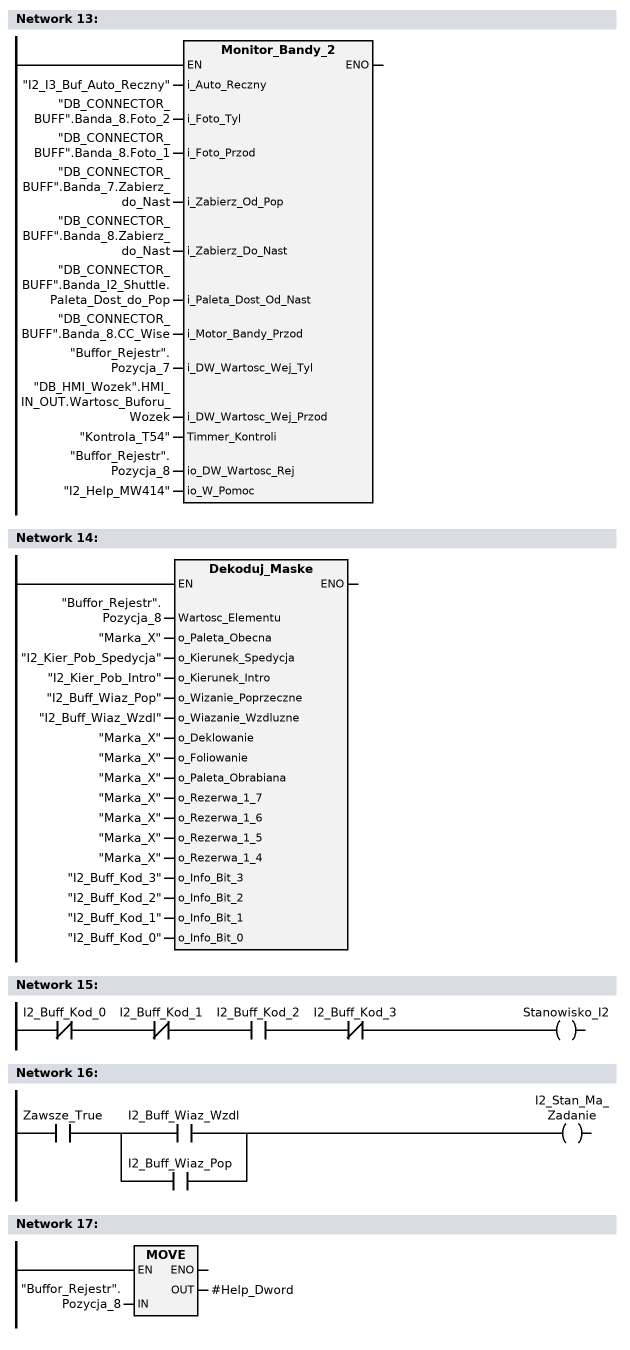
[picture p225: Stan_Intro_Pob_I2 networks 13-17]
NETWORK
TITLE =
//Monitoring band 8
//
      CALL  "Monitor_Bandy_2" (
           i_Auto_Reczny            := "I2_I3_Buf_Auto_Reczny",
           i_Foto_Tyl               := "DB_CONNECTOR_BUFF".Banda_8.Foto_2,
           i_Foto_Przod             := "DB_CONNECTOR_BUFF".Banda_8.Foto_1,
           i_Zabierz_Od_Pop         := "DB_CONNECTOR_BUFF".Banda_7.Zabierz_do_Nast,
           i_Zabierz_Do_Nast        := "DB_CONNECTOR_BUFF".Banda_8.Zabierz_do_Nast,
           i_Paleta_Dost_Od_Nast    := "DB_CONNECTOR_BUFF".Banda_I2_Shuttle.Paleta_Dost_do_Pop,
           i_Motor_Bandy_Przod      := "DB_CONNECTOR_BUFF".Banda_8.CC_Wise,
           i_DW_Wartosc_Wej_Tyl     := "Buffor_Rejestr".Pozycja_7,
           i_DW_Wartosc_Wej_Przod   := "DB_HMI_Wozek".HMI_IN_OUT.Wartosc_Buforu_Wozek,
           Timmer_Kontroli          := "Kontrola_T54",
           io_DW_Wartosc_Rej        := "Buffor_Rejestr".Pozycja_8,
           io_W_Pomoc               := "I2_Help_MW414");
NETWORK
TITLE =
//Dekouj maske
//Potrzebne do okreslenia kierunku kursu
      CALL  "Dekoduj_Maske" (
           Wartosc_Elementu         := "Buffor_Rejestr".Pozycja_8,
           o_Paleta_Obecna          := "Marka_X",
           o_Kierunek_Spedycja      := "I2_Kier_Pob_Spedycja",
           o_Kierunek_Intro         := "I2_Kier_Pob_Intro",
           o_Wizanie_Poprzeczne     := "I2_Buff_Wiaz_Pop",
           o_Wiazanie_Wzdluzne      := "I2_Buff_Wiaz_Wzdl",
           o_Deklowanie             := "Marka_X",
           o_Foliowanie             := "Marka_X",
           o_Paleta_Obrabiana       := "Marka_X",
           o_Rezerwa_1_7            := "Marka_X",
           o_Rezerwa_1_6            := "Marka_X",
           o_Rezerwa_1_5            := "Marka_X",
           o_Rezerwa_1_4            := "Marka_X",
           o_Info_Bit_3             := "I2_Buff_Kod_3",
           o_Info_Bit_2             := "I2_Buff_Kod_2",
           o_Info_Bit_1             := "I2_Buff_Kod_1",
           o_Info_Bit_0             := "I2_Buff_Kod_0");
NETWORK
TITLE =
//Stanowisko intro kod 
      AN    "I2_Buff_Kod_0";
      AN    "I2_Buff_Kod_1";
      A     "I2_Buff_Kod_2";
      AN    "I2_Buff_Kod_3";
      =     "Stanowisko_I2";
NETWORK
TITLE =
//Stanowisko intro ma jakies zadanie
      A     "Zawsze_True";
      A(;
      O     "I2_Buff_Wiaz_Wzdl";
      O     "I2_Buff_Wiaz_Pop";
      );
      =     "I2_Stan_Ma_Zadanie";
NETWORK
TITLE =
      L     "Buffor_Rejestr".Pozycja_8;
      T     #Help_Dword;
      NOP   0;
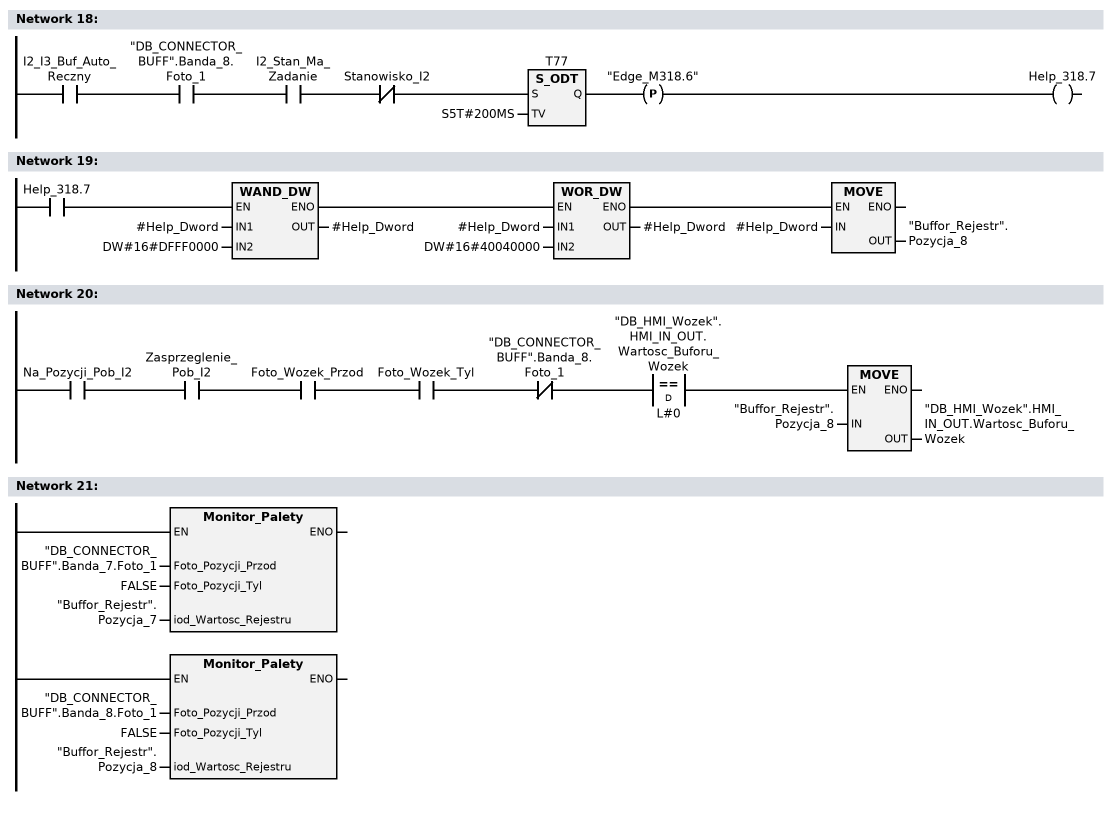
NETWORK
TITLE =
//Przepisanie wartosci nowej wartosci kodu jesli jest zadanie a paleta nie znana
//Domyslnie wysylana jest na Gender
      A(;
      A     "I2_I3_Buf_Auto_Reczny";
      A     "DB_CONNECTOR_BUFF".Banda_8.Foto_1;
      A     "I2_Stan_Ma_Zadanie";
      AN    "Stanowisko_I2";
      L     S5T#200MS;
      SD    "T77";
      NOP   0;
      NOP   0;
      NOP   0;
      A     "T77";
      );
      FP    "Edge_M318.6";
      =     "Help_318.7";
NETWORK
TITLE =
//Przypisanie nowej wartosci do palety
      A(;
      A(;
      A     "Help_318.7";
      JNB   _003;
      L     #Help_Dword;
      L     DW#16#DFFF0000;
      AD;
      T     #Help_Dword;
      SET;
      SAVE;
      CLR;
_003: A     BR;
      );
      JNB   _004;
      L     #Help_Dword;
      L     DW#16#40040000;
      OD;
      T     #Help_Dword;
      SET;
      SAVE;
      CLR;
_004: A     BR;
      );
      JNB   _005;
      L     #Help_Dword;
      T     "Buffor_Rejestr".Pozycja_8;
_005: NOP   0;
NETWORK
TITLE =
//db128.db208 -wartosc rejestru na wozka
      A     "Na_Pozycji_Pob_I2";
      A     "Zasprzeglenie_Pob_I2";
      A     "Foto_Wozek_Przod";
      A     "Foto_Wozek_Tyl";
      AN    "DB_CONNECTOR_BUFF".Banda_8.Foto_1;
      A(;
      L     "DB_HMI_Wozek".HMI_IN_OUT.Wartosc_Buforu_Wozek;
      L     L#0;
      ==D;
      );
      JNB   _006;
      L     "Buffor_Rejestr".Pozycja_8;
      T     "DB_HMI_Wozek".HMI_IN_OUT.Wartosc_Buforu_Wozek;
_006: NOP   0;
NETWORK
TITLE =
//Monitor palet
      CALL  "Monitor_Palety" (
           Foto_Pozycji_Przod       := "DB_CONNECTOR_BUFF".Banda_7.Foto_1,
           Foto_Pozycji_Tyl         := FALSE,
           iod_Wartosc_Rejestru     := "Buffor_Rejestr".Pozycja_7);
      CALL  "Monitor_Palety" (
           Foto_Pozycji_Przod       := "DB_CONNECTOR_BUFF".Banda_8.Foto_1,
           Foto_Pozycji_Tyl         := FALSE,
           iod_Wartosc_Rejestru     := "Buffor_Rejestr".Pozycja_8);
END_FUNCTION_BLOCK

FUNCTION_BLOCK "Stan_Intro_Pob_I3"	// FB 9
//Stanowisko intro Pobieranie
//Linia zlozona z 5 band odbierajacych
//
//
//B7 B8 BW
//===>
//
//2 Bandy kierunek zgodny
VERSION : 0.1
VAR
  Banda_17 : FB 33;
  Banda_18 : FB 33;
END_VAR
VAR_TEMP
  Help_Bit_1 : BOOL ;
  Help_Reczny : BOOL ;
  Help_int : INT ;
  Help_Dword : DWORD ;
  Help_INT_1 : DINT ;
END_VAR
BEGIN
NETWORK
TITLE =
//Ten Network celowo jest wolny
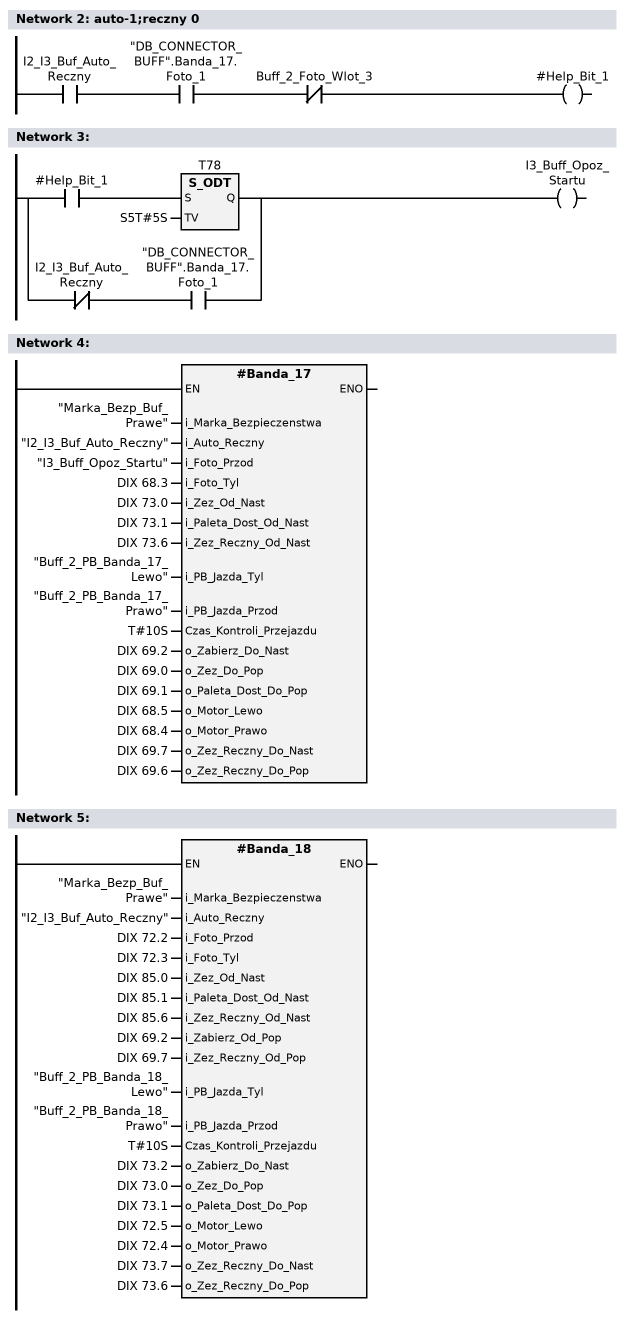
NETWORK
TITLE = auto-1;reczny 0
      A     "I2_I3_Buf_Auto_Reczny";
      A     "DB_CONNECTOR_BUFF".Banda_17.Foto_1;
      AN    "Buff_2_Foto_Wlot_3";
      =     #Help_Bit_1;
NETWORK
TITLE =
//Opoznienie startu po polozeniu palety
//
      O(;
      A     #Help_Bit_1;
      L     S5T#5S;
      SD    "T78";
      NOP   0;
      NOP   0;
      NOP   0;
      A     "T78";
      );
      O;
      AN    "I2_I3_Buf_Auto_Reczny";
      A     "DB_CONNECTOR_BUFF".Banda_17.Foto_1;
      =     "I3_Buff_Opoz_Startu";
NETWORK
TITLE =
//Banda 7
      CALL  #Banda_17 (
           i_Marka_Bezpieczenstwa   := "Marka_Bezp_Buf_Prawe",
           i_Auto_Reczny            := "I2_I3_Buf_Auto_Reczny",
           i_Foto_Przod             := "I3_Buff_Opoz_Startu",
           i_Foto_Tyl               := DIX 68.3,
           i_Zez_Od_Nast            := DIX 73.0,
           i_Paleta_Dost_Od_Nast    := DIX 73.1,
           i_Zez_Reczny_Od_Nast     := DIX 73.6,
           i_PB_Jazda_Tyl           := "Buff_2_PB_Banda_17_Lewo",
           i_PB_Jazda_Przod         := "Buff_2_PB_Banda_17_Prawo",
           Czas_Kontroli_Przejazdu  := T#10S,
           o_Zabierz_Do_Nast        := DIX 69.2,
           o_Zez_Do_Pop             := DIX 69.0,
           o_Paleta_Dost_Do_Pop     := DIX 69.1,
           o_Motor_Lewo             := DIX 68.5,
           o_Motor_Prawo            := DIX 68.4,
           o_Zez_Reczny_Do_Nast     := DIX 69.7,
           o_Zez_Reczny_Do_Pop      := DIX 69.6);
NETWORK
TITLE =
//Banda 8
      CALL  #Banda_18 (
           i_Marka_Bezpieczenstwa   := "Marka_Bezp_Buf_Prawe",
           i_Auto_Reczny            := "I2_I3_Buf_Auto_Reczny",
           i_Foto_Przod             := DIX 72.2,
           i_Foto_Tyl               := DIX 72.3,
           i_Zez_Od_Nast            := DIX 85.0,
           i_Paleta_Dost_Od_Nast    := DIX 85.1,
           i_Zez_Reczny_Od_Nast     := DIX 85.6,
           i_Zabierz_Od_Pop         := DIX 69.2,
           i_Zez_Reczny_Od_Pop      := DIX 69.7,
           i_PB_Jazda_Tyl           := "Buff_2_PB_Banda_18_Lewo",
           i_PB_Jazda_Przod         := "Buff_2_PB_Banda_18_Prawo",
           Czas_Kontroli_Przejazdu  := T#10S,
           o_Zabierz_Do_Nast        := DIX 73.2,
           o_Zez_Do_Pop             := DIX 73.0,
           o_Paleta_Dost_Do_Pop     := DIX 73.1,
           o_Motor_Lewo             := DIX 72.5,
           o_Motor_Prawo            := DIX 72.4,
           o_Zez_Reczny_Do_Nast     := DIX 73.7,
           o_Zez_Reczny_Do_Pop      := DIX 73.6);
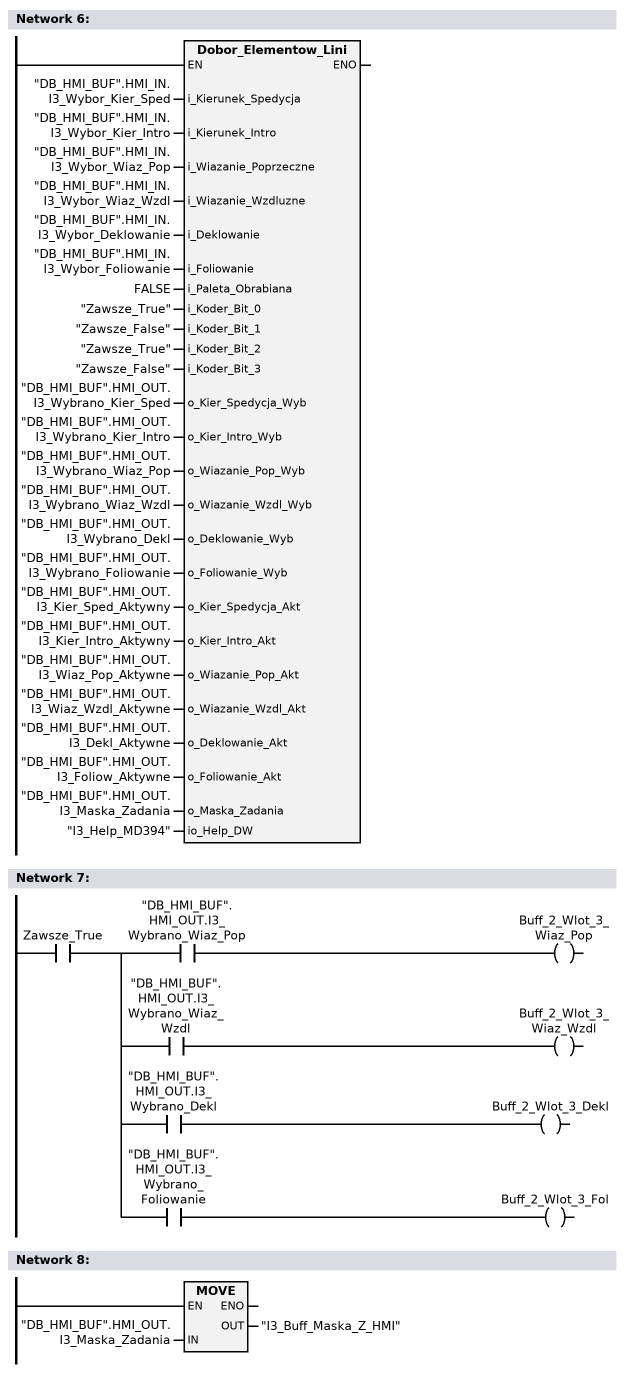
NETWORK
TITLE =
//Wybor Elementow na lini koder nr 5
      CALL  "Dobor_Elementow_Lini" (
           i_Kierunek_Spedycja      := "DB_HMI_BUF".HMI_IN.I3_Wybor_Kier_Sped,
           i_Kierunek_Intro         := "DB_HMI_BUF".HMI_IN.I3_Wybor_Kier_Intro,
           i_Wiazanie_Poprzeczne    := "DB_HMI_BUF".HMI_IN.I3_Wybor_Wiaz_Pop,
           i_Wiazanie_Wzdluzne      := "DB_HMI_BUF".HMI_IN.I3_Wybor_Wiaz_Wzdl,
           i_Deklowanie             := "DB_HMI_BUF".HMI_IN.I3_Wybor_Deklowanie,
           i_Foliowanie             := "DB_HMI_BUF".HMI_IN.I3_Wybor_Foliowanie,
           i_Paleta_Obrabiana       := FALSE,
           i_Koder_Bit_0            := "Zawsze_True",
           i_Koder_Bit_1            := "Zawsze_False",
           i_Koder_Bit_2            := "Zawsze_True",
           i_Koder_Bit_3            := "Zawsze_False",
           o_Kier_Spedycja_Wyb      := "DB_HMI_BUF".HMI_OUT.I3_Wybrano_Kier_Sped,
           o_Kier_Intro_Wyb         := "DB_HMI_BUF".HMI_OUT.I3_Wybrano_Kier_Intro,
           o_Wiazanie_Pop_Wyb       := "DB_HMI_BUF".HMI_OUT.I3_Wybrano_Wiaz_Pop,
           o_Wiazanie_Wzdl_Wyb      := "DB_HMI_BUF".HMI_OUT.I3_Wybrano_Wiaz_Wzdl,
           o_Deklowanie_Wyb         := "DB_HMI_BUF".HMI_OUT.I3_Wybrano_Dekl,
           o_Foliowanie_Wyb         := "DB_HMI_BUF".HMI_OUT.I3_Wybrano_Foliowanie,
           o_Kier_Spedycja_Akt      := "DB_HMI_BUF".HMI_OUT.I3_Kier_Sped_Aktywny,
           o_Kier_Intro_Akt         := "DB_HMI_BUF".HMI_OUT.I3_Kier_Intro_Aktywny,
           o_Wiazanie_Pop_Akt       := "DB_HMI_BUF".HMI_OUT.I3_Wiaz_Pop_Aktywne,
           o_Wiazanie_Wzdl_Akt      := "DB_HMI_BUF".HMI_OUT.I3_Wiaz_Wzdl_Aktywne,
           o_Deklowanie_Akt         := "DB_HMI_BUF".HMI_OUT.I3_Dekl_Aktywne,
           o_Foliowanie_Akt         := "DB_HMI_BUF".HMI_OUT.I3_Foliow_Aktywne,
           o_Maska_Zadania          := "DB_HMI_BUF".HMI_OUT.I3_Maska_Zadania,
           io_Help_DW               := "I3_Help_MD394");
NETWORK
TITLE =
//Wyswietlenie lampek zadania lini
      A     "Zawsze_True";
      =     L 12.0;
      A     L 12.0;
      A     "DB_HMI_BUF".HMI_OUT.I3_Wybrano_Wiaz_Pop;
      =     "Buff_2_Wlot_3_Wiaz_Pop";
      A     L 12.0;
      A     "DB_HMI_BUF".HMI_OUT.I3_Wybrano_Wiaz_Wzdl;
      =     "Buff_2_Wlot_3_Wiaz_Wzdl";
      A     L 12.0;
      A     "DB_HMI_BUF".HMI_OUT.I3_Wybrano_Dekl;
      =     "Buff_2_Wlot_3_Dekl";
      A     L 12.0;
      A     "DB_HMI_BUF".HMI_OUT.I3_Wybrano_Foliowanie;
      =     "Buff_2_Wlot_3_Fol";
NETWORK
TITLE =
//Przypisanie maski zadania do bandy wejsciowej
      L     "DB_HMI_BUF".HMI_OUT.I3_Maska_Zadania;
      T     "I3_Buff_Maska_Z_HMI";
      NOP   0;
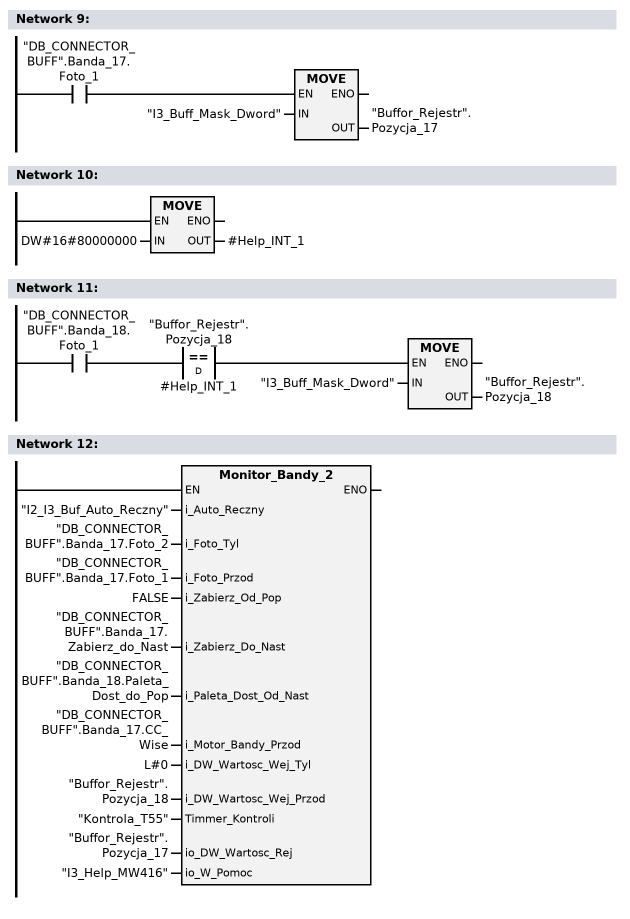
NETWORK
TITLE =
//Zbudowanie z maski podwojnego slowa
      A     "DB_CONNECTOR_BUFF".Banda_17.Foto_1;
      JNB   _001;
      L     "I3_Buff_Mask_Dword";
      T     "Buffor_Rejestr".Pozycja_17;
_001: NOP   0;
NETWORK
TITLE =
      L     DW#16#80000000;
      T     #Help_INT_1;
      NOP   0;
NETWORK
TITLE =
//sprawdzenie dla fotokomorki bandy 8
      A     "DB_CONNECTOR_BUFF".Banda_18.Foto_1;
      A(;
      L     "Buffor_Rejestr".Pozycja_18;
      L     #Help_INT_1;
      ==D;
      );
      JNB   _002;
      L     "I3_Buff_Mask_Dword";
      T     "Buffor_Rejestr".Pozycja_18;
_002: NOP   0;
NETWORK
TITLE =
//Monitoring band 7
      CALL  "Monitor_Bandy_2" (
           i_Auto_Reczny            := "I2_I3_Buf_Auto_Reczny",
           i_Foto_Tyl               := "DB_CONNECTOR_BUFF".Banda_17.Foto_2,
           i_Foto_Przod             := "DB_CONNECTOR_BUFF".Banda_17.Foto_1,
           i_Zabierz_Od_Pop         := FALSE,
           i_Zabierz_Do_Nast        := "DB_CONNECTOR_BUFF".Banda_17.Zabierz_do_Nast,
           i_Paleta_Dost_Od_Nast    := "DB_CONNECTOR_BUFF".Banda_18.Paleta_Dost_do_Pop,
           i_Motor_Bandy_Przod      := "DB_CONNECTOR_BUFF".Banda_17.CC_Wise,
           i_DW_Wartosc_Wej_Tyl     := L#0,
           i_DW_Wartosc_Wej_Przod   := "Buffor_Rejestr".Pozycja_18,
           Timmer_Kontroli          := "Kontrola_T55",
           io_DW_Wartosc_Rej        := "Buffor_Rejestr".Pozycja_17,
           io_W_Pomoc               := "I3_Help_MW416");
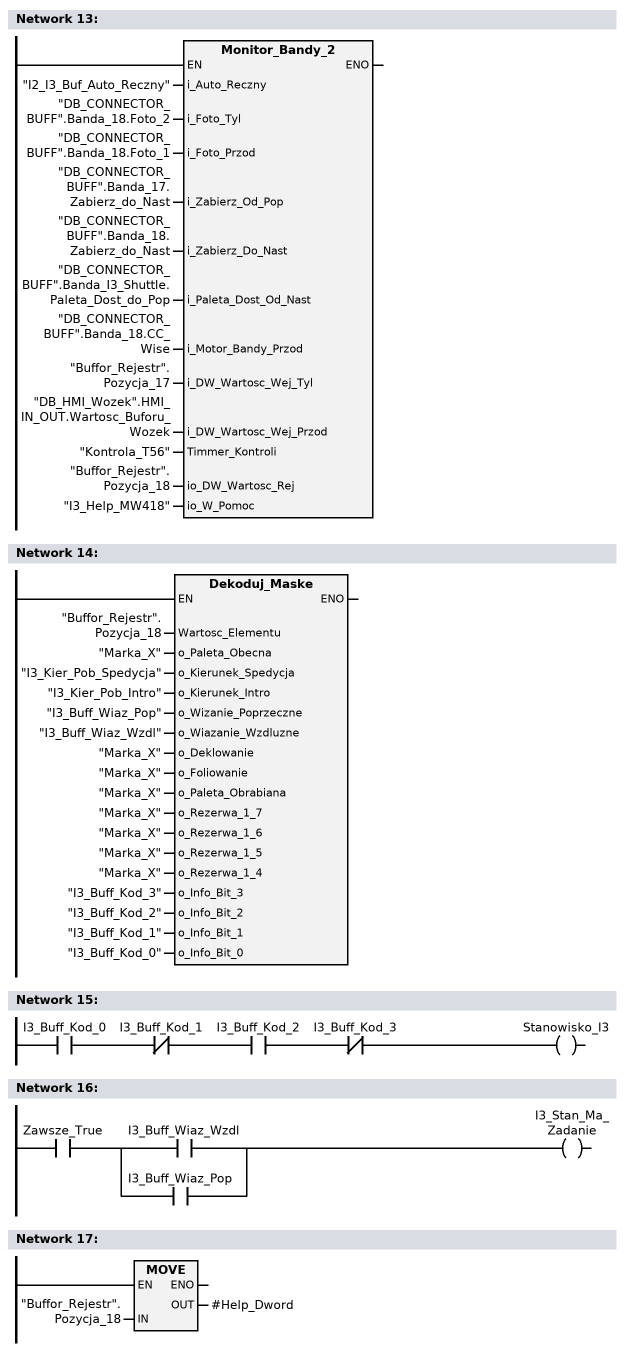
NETWORK
TITLE =
//Monitoring band 8
//
      CALL  "Monitor_Bandy_2" (
           i_Auto_Reczny            := "I2_I3_Buf_Auto_Reczny",
           i_Foto_Tyl               := "DB_CONNECTOR_BUFF".Banda_18.Foto_2,
           i_Foto_Przod             := "DB_CONNECTOR_BUFF".Banda_18.Foto_1,
           i_Zabierz_Od_Pop         := "DB_CONNECTOR_BUFF".Banda_17.Zabierz_do_Nast,
           i_Zabierz_Do_Nast        := "DB_CONNECTOR_BUFF".Banda_18.Zabierz_do_Nast,
           i_Paleta_Dost_Od_Nast    := "DB_CONNECTOR_BUFF".Banda_I3_Shuttle.Paleta_Dost_do_Pop,
           i_Motor_Bandy_Przod      := "DB_CONNECTOR_BUFF".Banda_18.CC_Wise,
           i_DW_Wartosc_Wej_Tyl     := "Buffor_Rejestr".Pozycja_17,
           i_DW_Wartosc_Wej_Przod   := "DB_HMI_Wozek".HMI_IN_OUT.Wartosc_Buforu_Wozek,
           Timmer_Kontroli          := "Kontrola_T56",
           io_DW_Wartosc_Rej        := "Buffor_Rejestr".Pozycja_18,
           io_W_Pomoc               := "I3_Help_MW418");
NETWORK
TITLE =
//Dekouj maske
//Potrzebne do okreslenia kierunku kursu
      CALL  "Dekoduj_Maske" (
           Wartosc_Elementu         := "Buffor_Rejestr".Pozycja_18,
           o_Paleta_Obecna          := "Marka_X",
           o_Kierunek_Spedycja      := "I3_Kier_Pob_Spedycja",
           o_Kierunek_Intro         := "I3_Kier_Pob_Intro",
           o_Wizanie_Poprzeczne     := "I3_Buff_Wiaz_Pop",
           o_Wiazanie_Wzdluzne      := "I3_Buff_Wiaz_Wzdl",
           o_Deklowanie             := "Marka_X",
           o_Foliowanie             := "Marka_X",
           o_Paleta_Obrabiana       := "Marka_X",
           o_Rezerwa_1_7            := "Marka_X",
           o_Rezerwa_1_6            := "Marka_X",
           o_Rezerwa_1_5            := "Marka_X",
           o_Rezerwa_1_4            := "Marka_X",
           o_Info_Bit_3             := "I3_Buff_Kod_3",
           o_Info_Bit_2             := "I3_Buff_Kod_2",
           o_Info_Bit_1             := "I3_Buff_Kod_1",
           o_Info_Bit_0             := "I3_Buff_Kod_0");
NETWORK
TITLE =
//Stanowisko intro kod 
      A     "I3_Buff_Kod_0";
      AN    "I3_Buff_Kod_1";
      A     "I3_Buff_Kod_2";
      AN    "I3_Buff_Kod_3";
      =     "Stanowisko_I3";
NETWORK
TITLE =
//Stanowisko intro ma jakies zadanie
      A     "Zawsze_True";
      A(;
      O     "I3_Buff_Wiaz_Wzdl";
      O     "I3_Buff_Wiaz_Pop";
      );
      =     "I3_Stan_Ma_Zadanie";
NETWORK
TITLE =
      L     "Buffor_Rejestr".Pozycja_18;
      T     #Help_Dword;
      NOP   0;
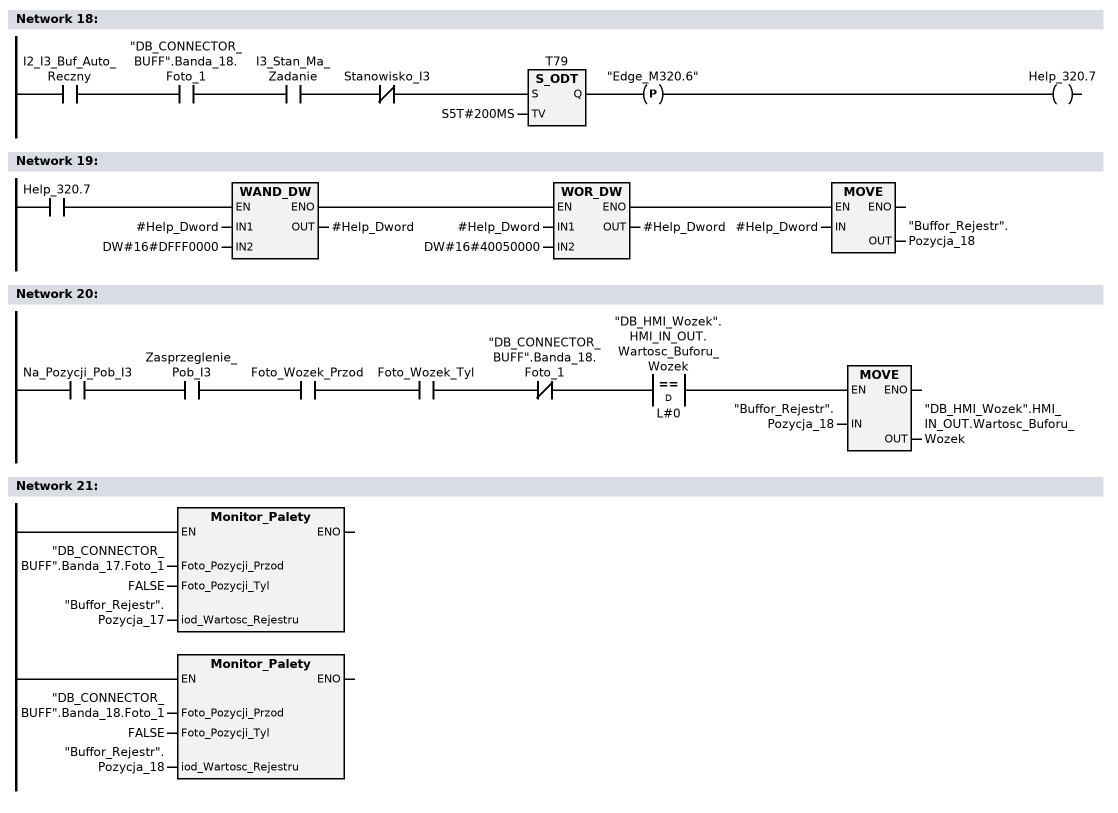
NETWORK
TITLE =
//Przepisanie wartosci nowej wartosci kodu jesli jest zadanie a paleta nie znana
//Domyslnie wysylana jest na Gender
      A(;
      A     "I2_I3_Buf_Auto_Reczny";
      A     "DB_CONNECTOR_BUFF".Banda_18.Foto_1;
      A     "I3_Stan_Ma_Zadanie";
      AN    "Stanowisko_I3";
      L     S5T#200MS;
      SD    "T79";
      NOP   0;
      NOP   0;
      NOP   0;
      A     "T79";
      );
      FP    "Edge_M320.6";
      =     "Help_320.7";
NETWORK
TITLE =
//Przypisanie nowej wartosci do palety
      A(;
      A(;
      A     "Help_320.7";
      JNB   _003;
      L     #Help_Dword;
      L     DW#16#DFFF0000;
      AD;
      T     #Help_Dword;
      SET;
      SAVE;
      CLR;
_003: A     BR;
      );
      JNB   _004;
      L     #Help_Dword;
      L     DW#16#40050000;
      OD;
      T     #Help_Dword;
      SET;
      SAVE;
      CLR;
_004: A     BR;
      );
      JNB   _005;
      L     #Help_Dword;
      T     "Buffor_Rejestr".Pozycja_18;
_005: NOP   0;
NETWORK
TITLE =
//db128.db208 -wartosc rejestru na wozka
      A     "Na_Pozycji_Pob_I3";
      A     "Zasprzeglenie_Pob_I3";
      A     "Foto_Wozek_Przod";
      A     "Foto_Wozek_Tyl";
      AN    "DB_CONNECTOR_BUFF".Banda_18.Foto_1;
      A(;
      L     "DB_HMI_Wozek".HMI_IN_OUT.Wartosc_Buforu_Wozek;
      L     L#0;
      ==D;
      );
      JNB   _006;
      L     "Buffor_Rejestr".Pozycja_18;
      T     "DB_HMI_Wozek".HMI_IN_OUT.Wartosc_Buforu_Wozek;
_006: NOP   0;
NETWORK
TITLE =
//Monitor palet
      CALL  "Monitor_Palety" (
           Foto_Pozycji_Przod       := "DB_CONNECTOR_BUFF".Banda_17.Foto_1,
           Foto_Pozycji_Tyl         := FALSE,
           iod_Wartosc_Rejestru     := "Buffor_Rejestr".Pozycja_17);
      CALL  "Monitor_Palety" (
           Foto_Pozycji_Przod       := "DB_CONNECTOR_BUFF".Banda_18.Foto_1,
           Foto_Pozycji_Tyl         := FALSE,
           iod_Wartosc_Rejestru     := "Buffor_Rejestr".Pozycja_18);
END_FUNCTION_BLOCK

FUNCTION_BLOCK "FB_Uzbrajanie"	// FB 10
//Funkcja odpowiada za sterowanie uzbrajaniem palety.
//Gdy jest stan wysoki na wejsciu uzbrajanie palety to aktywne jest przycisk 
//PB_uzbrajanie (Pojedyncze klikniecie). Aby zakonczyc uzbrajanie nalezy wcisnac 
//przycisk dwukrotnie w krotkim czasie.
VERSION : 0.1
VAR_INPUT
  i_Tryb_Uzbrajania : BOOL ;
  i_Zezw_Na_Uzb : BOOL ;	//Zezwolenie na uzbrajanie
  i_PB_Uzbrajanie : BOOL ;	//Przycisk grzybkowy uzbrajania
  i_PB_Wybor_O_Lewo : BOOL ;	//Wybor obrot w lewa strone
  i_PB_Wybor_O_Prawo : BOOL ;	//Wybor obrot w prawa strone
  i_Pedal_Zal : BOOL ;	//Wlaczenie pedala
  t_Czas_Kontrolny : TIME ;
  t_Czas_Konca : TIME ;
END_VAR
VAR_OUTPUT
  o_Oczekiwanie_Aktywne : BOOL ;
  o_Lampka_Uzb_Lewo : BOOL ;
  o_Lampka_Uzb_Prawo : BOOL ;
  o_Sygnal_Startu_Uzbr : BOOL ;	//Sygnal krotki startu uzbrajania
  o_Sygnal_Kon_Uzbr : BOOL ;	//Sygnal konca uzbrajania
  o_Pedal_Lewo : BOOL ;
  o_Pedal_Prawo : BOOL ;
END_VAR
VAR_IN_OUT
  io_Uzbrajanie_W_Trakcie : BOOL ;
END_VAR
VAR
  Czas_Kontrolny : SFB 4;	//Czas kontrolny przycisku
  Czas_Konca : SFB 4;
  Edge_1 : BOOL ;
  Edge_2 : BOOL ;
  Edge_3 : BOOL ;
  Help_Timer : BOOL ;
  H_Uzbrajanie_W_Trakcie : BOOL ;
  H_Lewo_Prawo : BOOL ;	//0-Lewo;1-Prawo
END_VAR
VAR_TEMP
  Temp_Bit_1 : BOOL ;
  Temp_Bit_2 : BOOL ;
END_VAR
BEGIN
NETWORK
TITLE =
//Ten Network celowo jest wolny
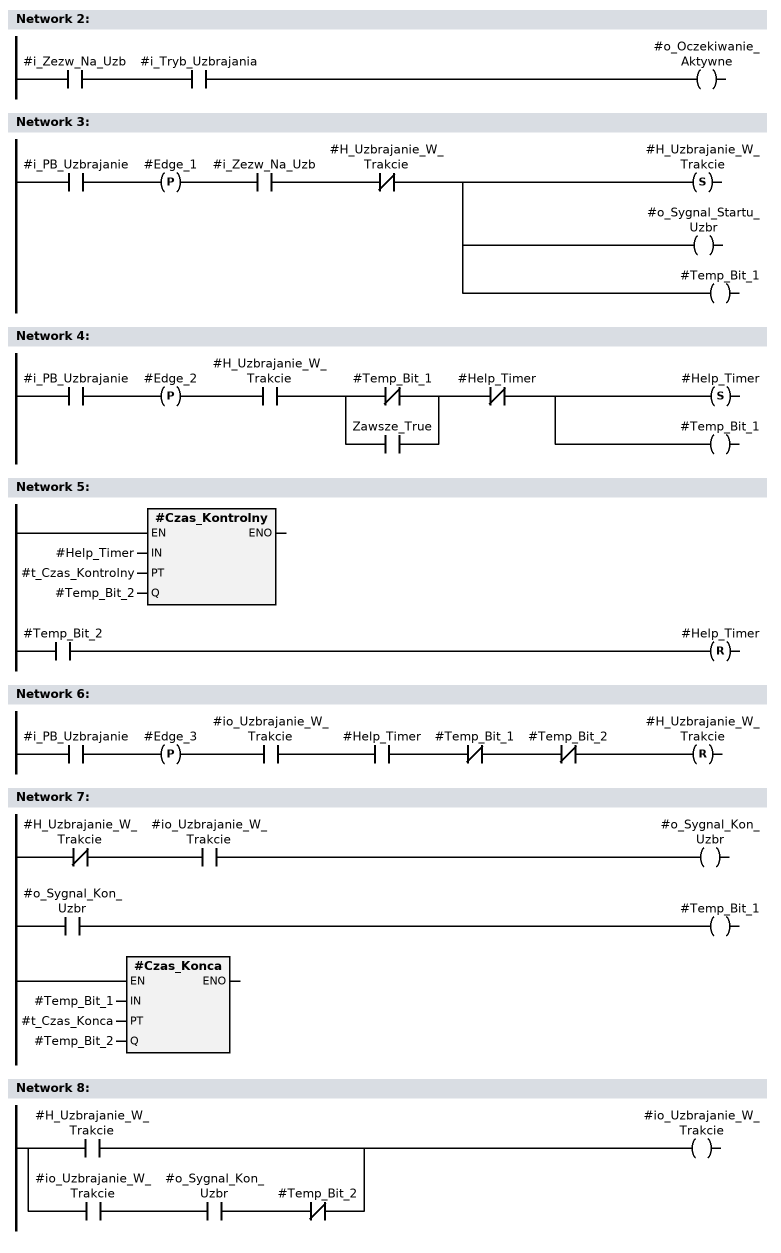
NETWORK
TITLE =
//Informacja ze czeka na sygnal uzbrajania.Gdy jest oczekiwanie powinna migac 
//lampka (np ¿ó³ta)
      A     #i_Zezw_Na_Uzb;
      A     #i_Tryb_Uzbrajania;
      =     #o_Oczekiwanie_Aktywne;
NETWORK
TITLE =
//Uzbrajanie jest aktyne
      A     #i_PB_Uzbrajanie;
      FP    #Edge_1;
      A     #i_Zezw_Na_Uzb;
      AN    #H_Uzbrajanie_W_Trakcie;
      S     #H_Uzbrajanie_W_Trakcie;
      =     #o_Sygnal_Startu_Uzbr;
      =     #Temp_Bit_1;
NETWORK
TITLE =
//kasowanie uzbrajania palety
//Temp_Bit_1 wykorzystany pare networkow dalej
      A     #i_PB_Uzbrajanie;
      FP    #Edge_2;
      A     #H_Uzbrajanie_W_Trakcie;
      A(;
      ON    #Temp_Bit_1;
      O     "Zawsze_True";
      );
      AN    #Help_Timer;
      S     #Help_Timer;
      =     #Temp_Bit_1;
NETWORK
TITLE =
//Timer kontrolny realizujacy funkcje wylaczenia uzbrajania palety
      CALL  #Czas_Kontrolny (
           IN                       := #Help_Timer,
           PT                       := #t_Czas_Kontrolny,
           Q                        := #Temp_Bit_2);
      A     #Temp_Bit_2;
//Resetowanie Timmera
      R     #Help_Timer;
NETWORK
TITLE =
//Resetowanie uzbrajania
      A     #i_PB_Uzbrajanie;
      FP    #Edge_3;
      A     #io_Uzbrajanie_W_Trakcie;
      A     #Help_Timer;
      AN    #Temp_Bit_1;
      AN    #Temp_Bit_2;
      R     #H_Uzbrajanie_W_Trakcie;
NETWORK
TITLE =
//Sygnal konca uzbrajania
      AN    #H_Uzbrajanie_W_Trakcie;
      A     #io_Uzbrajanie_W_Trakcie;
      =     #o_Sygnal_Kon_Uzbr;
      A     #o_Sygnal_Kon_Uzbr;
      =     #Temp_Bit_1;
      CALL  #Czas_Konca (
           IN                       := #Temp_Bit_1,
           PT                       := #t_Czas_Konca,
           Q                        := #Temp_Bit_2);
NETWORK
TITLE =
//Podtrzymanie do zakonczenia
      O     #H_Uzbrajanie_W_Trakcie;
      O;
      A     #io_Uzbrajanie_W_Trakcie;
      A     #o_Sygnal_Kon_Uzbr;
      AN    #Temp_Bit_2;
      =     #io_Uzbrajanie_W_Trakcie;
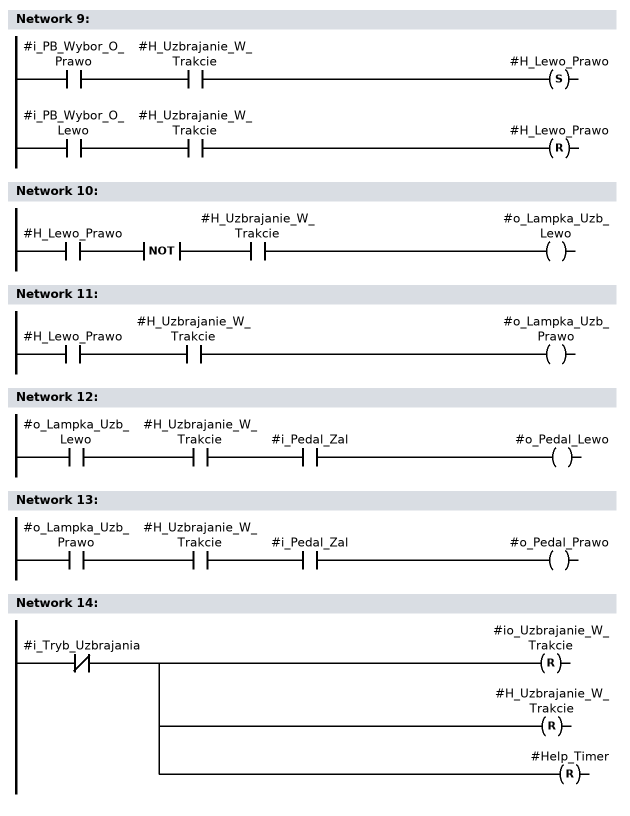
NETWORK
TITLE =
//Przyciski zmiany kierunku owijania
//
      A     #i_PB_Wybor_O_Prawo;
      A     #H_Uzbrajanie_W_Trakcie;
      S     #H_Lewo_Prawo;
      A     #i_PB_Wybor_O_Lewo;
      A     #H_Uzbrajanie_W_Trakcie;
      R     #H_Lewo_Prawo;
      NOP   0;
NETWORK
TITLE =
//Lampka lewo
      A     #H_Lewo_Prawo;
      NOT;
      A     #H_Uzbrajanie_W_Trakcie;
      =     #o_Lampka_Uzb_Lewo;
NETWORK
TITLE =
//Lampka prawo
      A     #H_Lewo_Prawo;
      A     #H_Uzbrajanie_W_Trakcie;
      =     #o_Lampka_Uzb_Prawo;
NETWORK
TITLE =
//Jazda lewo
//
      A     #o_Lampka_Uzb_Lewo;
      A     #H_Uzbrajanie_W_Trakcie;
      A     #i_Pedal_Zal;
      =     #o_Pedal_Lewo;
NETWORK
TITLE =
//Jazda lewo
//
      A     #o_Lampka_Uzb_Prawo;
      A     #H_Uzbrajanie_W_Trakcie;
      A     #i_Pedal_Zal;
      =     #o_Pedal_Prawo;
NETWORK
TITLE =
      AN    #i_Tryb_Uzbrajania;
      R     #io_Uzbrajanie_W_Trakcie;
      R     #H_Uzbrajanie_W_Trakcie;
      R     #Help_Timer;
END_FUNCTION_BLOCK

FUNCTION_BLOCK "T_ON"	// FB 20
//Funkcja zatrzymujaca czas gdy na wejsciu stop pojawi sie stan niski. Wartosc 
//wejscia TON nie jest wtedy brana pod uwage. 
AUTHOR : Kng
NAME : Help_FB
VERSION : 0.1
VAR_INPUT
  IN : BOOL ;	//Wejscie aktywujace timer
  STOP : BOOL ;	//Sygnal aktywny stanem wysokim
  PT : TIME ;	//Czas zadany
END_VAR
VAR_OUTPUT
  Q_0 : BOOL ;
END_VAR
VAR_IN_OUT
  ET : TIME ;
END_VAR
VAR
  T_1 : SFB 4;
  Help_Zbocze_1 : BOOL ;
  Help_Zbocze_2 : BOOL ;
  Help_Zbocze_3 : BOOL ;
END_VAR
BEGIN
NETWORK
TITLE =
//Ten network celowo jest wolny
NETWORK
TITLE =
// Zapisanie wartosci czasu w pamieci
      A     #STOP;
      FN    #Help_Zbocze_1;
      A     #IN;
      JCN   et_1;
      L     #T_1.PT;
      L     #T_1.ET;
      -D;
      T     #T_1.PT;
      SET;
      R     #T_1.IN;
et_1: NOP   0;
//Przywrocenie czasu zapisanego
      A     #STOP;
      FP    #Help_Zbocze_2;
      A     #IN;
      S     #T_1.IN;
//Warunki poczatkowe
      A     #IN;
      FP    #Help_Zbocze_3;
      A     #STOP;
      JCN   et_3;
      L     #PT;
      T     #T_1.PT;
      SET;
      S     #T_1.IN;
et_3: NOP   0;
//Wywolaj funkcje timera
      CALL  #T_1;
      A     #T_1.Q;
      S     #Q_0;
      AN    #IN;
      A     #STOP;
//Wystaw wyjscie gdy skonczy sie czas
      R     #T_1.IN;
      R     #Q_0;
      L     #T_1.PT;
      L     #T_1.ET;
      -D;
      T     #ET;
//Pokaz wartosc czasu
END_FUNCTION_BLOCK

FUNCTION_BLOCK "T_ON_+_RESET"	// FB 21
//Funkcja zatrzymujaca czas gdy na wejsciu stop pojawi sie stan niski. Wartosc 
//wejscia TON nie jest wtedy brana pod uwage. 
//Dodano przycisk reset.
AUTHOR : Kng
NAME : Help_FB
VERSION : 1.1
VAR_INPUT
  IN : BOOL ;	//Wejscie aktywujace timer
  STOP : BOOL ;	//Sygnal aktywny stanem wysokim
  PT : TIME ;	//Czas zadany
  RESET : BOOL ;	//Wejescie resetujace aktywne stanem wysokim
END_VAR
VAR_OUTPUT
  Q_0 : BOOL ;
END_VAR
VAR_IN_OUT
  ET : TIME ;
END_VAR
VAR
  T_1 : SFB 4;
  Help_Zbocze_1 : BOOL ;
  Help_Zbocze_2 : BOOL ;
  Help_Zbocze_3 : BOOL ;
  Help_Zbocze_4 : BOOL ;
  Help_Zbocze_5 : BOOL ;
END_VAR
BEGIN
NETWORK
TITLE =
//Ten network celowo jest wolny
NETWORK
TITLE =
      A     #RESET;
      S     #Help_Zbocze_4;
// Zapisanie wartosci czasu w pamieci
      A     #STOP;
      FN    #Help_Zbocze_1;
      A     #IN;
      JCN   et_2;
      L     #T_1.PT;
      L     #T_1.ET;
      -D;
      T     #T_1.PT;
      SET;
      R     #T_1.IN;
et_2: NOP   0;
//Przywrocenie czasu zapisanego
      A     #STOP;
      FP    #Help_Zbocze_2;
      A     #IN;
      S     #T_1.IN;
//Wystaw wyjscie gdy skonczy sie czas
      A     #T_1.Q;
      S     #Q_0;
      AN    #IN;
      A     #STOP;
      O;
      A     #RESET;
      R     #T_1.IN;
      R     #Q_0;
//Warunki poczatkowe  oraz reset
      AN    #RESET;
      A     #Help_Zbocze_4;
      O;
      A(;
      A     #IN;
      FP    #Help_Zbocze_3;
      A     #STOP;
      );
      JCN   et_3;
      L     #PT;
      T     #T_1.PT;
      SET;
      R     #Help_Zbocze_4;
//brak wysterownia jezeli reset robiony bez stopu
      A     #STOP;
      S     #T_1.IN;
et_3: NOP   0;
//Wywolaj funkcje timera
      CALL  #T_1;
      L     #T_1.PT;
      L     #T_1.ET;
      -D;
      T     #ET;
//Pokaz wartosc czasu
END_FUNCTION_BLOCK

FUNCTION_BLOCK "Band_Wozka"	// FB 32
//Funkcja realizujaca koncepcje bandy pojedycznej, ktora uwzglednia rowniez tryb 
//reczny. W celu lepszego sterowania trybem recznym nalezy do³o¿yæ:
//-fotokomorki na tyle bandy.
//-fotokomorka na tyle okresla rowniez zajetosc
//-jazda do tylu bandy mozliwa
//-jazda do przodu poza fotokomorke mozliwa gdy nastepna w ruchu i wolna.
//-do³o¿enie okresnia trybu reczny/auto gdzie auto to 1 
//
AUTHOR : Kng
FAMILY : Bandy
NAME : B_Single
VERSION : 1.0
VAR_INPUT
  i_Marka_Bezpieczenstwa : BOOL ;
  i_Odwrocenie : BOOL ;	//Wejscie odwracajaca dzialanie bandy
  i_Auto_Reczny : BOOL ;	//1-auto,0-reczny
  i_Foto_Przod : BOOL ;	//Foto na koncu tasmy
  i_Foto_Tyl : BOOL ;	//Foto zapobiegajace wyjechaniu palety do tylu
  i_Zez_Od_Nast : BOOL ;
  i_Paleta_Dost_Od_Nast : BOOL ;
  i_Zez_Reczny_Od_Nast : BOOL ;
  i_Zabierz_Od_Pop : BOOL ;
  i_Zez_Reczny_Od_Pop : BOOL ;
  i_PB_Jazda_Tyl : BOOL ;
  i_PB_Jazda_Przod : BOOL ;
  i_Reset_Interfejsu : BOOL ;	//Reset interfejsu
  Czas_Kontroli_Przejazdu : TIME ;
END_VAR
VAR_OUTPUT
  o_Zabierz_Do_Nast : BOOL ;	//Rozkaz pobrania do nast bandy
  o_Zez_Do_Pop : BOOL ;
  o_Paleta_Dost_Do_Pop : BOOL ;
  o_Motor_Lewo : BOOL ;
  o_Motor_Prawo : BOOL ;
  o_Zez_Reczny_Do_Nast : BOOL ;
  o_Zez_Reczny_Do_Pop : BOOL ;
  o_Zajetosc_Nieb : BOOL ;	//Dla bezpieczenstwa transportu
END_VAR
VAR
  Czas_kontrolny : FB 20;
  Help_A_Motor_Lewo : BOOL ;
  S_Help_Zab_Od_Pop : BOOL ;
  Stop_Czas_Kontrolny : BOOL ;
  Zbocze_1 : BOOL ;
  Zbocze_2 : BOOL ;
  Blokada_Wjazdu : BOOL ;
  Help_H_Motor_Prawo : BOOL ;
  Help_H_Motor_Lewo : BOOL ;
  Toggle : BOOL ;	//bit przemienny dla auto i hand
  H_Foto_Przod : BOOL ;
  H_Foto_Tyl : BOOL ;
  H_o_Zez_Do_Pop : BOOL ;
  H_o_Zabierz_Do_Nast : BOOL ;
  H3 : BOOL ;
  H4 : BOOL ;
  H5 : BOOL ;
  H6 : BOOL ;
  Czas_Opoz_1 : FB 20;
  Czas_Opoz_2 : FB 20;
  Czas_Opoz_3 : FB 20;
  Czas_Opoz_4 : FB 20;
  Czas_Opoz_5 : FB 20;
END_VAR
VAR_TEMP
  Temp_Help_1 : BOOL ;
  Temp_Help_2 : BOOL ;
  Czas_zadany : TIME ;
  Czas_aktualny : TIME ;
  Temp_Help_3 : BOOL ;
  Temp_Help_4 : BOOL ;
END_VAR
BEGIN
NETWORK
TITLE =
//
// B1        B2         foto_1    foto_2         B5        B6
//(\\\\\\\\\\\\\\\\\\)  (\\\\\\\\\\\\\\\\\\)  (\\\\\\\\\\\\\\\\\\)
//                  M1                    M2                     M3
//         
//        zabierz <-- pobierz      |  zabierz    <--  pobierz  
//     zez_do_pop --> zez_od_nast  |  zez_od_pop -->  zez_od_nast
//                                  
//-Uklad dzielony jest na realizowane funkcje
//
//         <----------------------------------------- kierunek
//                  
//
// ten network celowo jest pusty
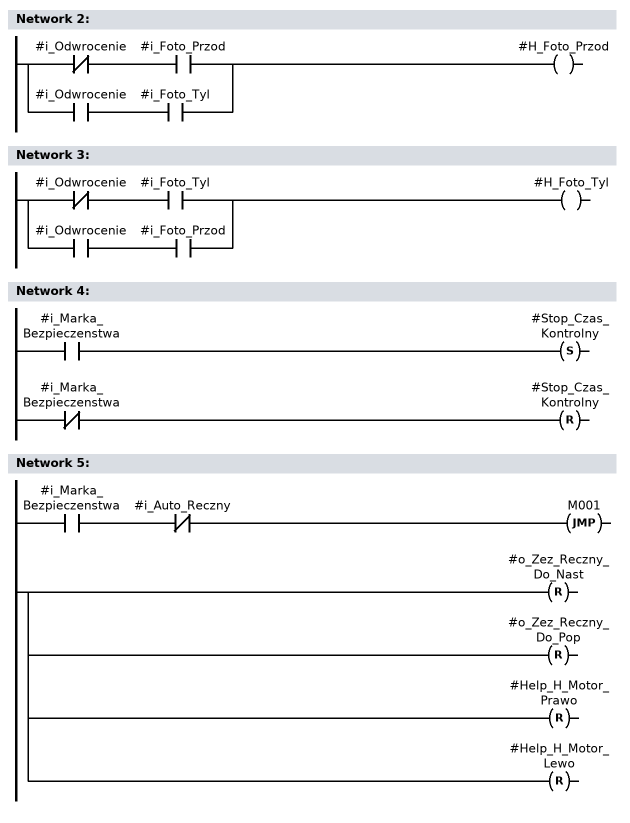
NETWORK
TITLE =
//Odwrocenie sygnalow fotokomorek
      AN    #i_Odwrocenie;
      A     #i_Foto_Przod;
      O;
      A     #i_Odwrocenie;
      A     #i_Foto_Tyl;
      =     #H_Foto_Przod;
NETWORK
TITLE =
//Odwrocenie sygnalow fotokomorek
      AN    #i_Odwrocenie;
      A     #i_Foto_Tyl;
      O;
      A     #i_Odwrocenie;
      A     #i_Foto_Przod;
      =     #H_Foto_Tyl;
NETWORK
TITLE =
//Sprawdzenie stanu bezpieczenstwa lub freeze
//Skocz jezeli brak marki bezpieczenstwa
//Marka bezpieczenstwa ok gdy wysoki
      A     #i_Marka_Bezpieczenstwa;
      S     #Stop_Czas_Kontrolny;
//      AN    #i_Marka_Bezpieczenstwa
//      AN    #Stop_Czas_Kontrolny
//      JC    end
      AN    #i_Marka_Bezpieczenstwa;
      R     #Stop_Czas_Kontrolny;
NETWORK
TITLE =
//Wyznczenie zbocza pozytywnego i negatywnego
//skok do trybu recznego 
      A     #i_Marka_Bezpieczenstwa;
      AN    #i_Auto_Reczny;
      JC    M001;
//czyszczenie trybu recznego
      SET;
      R     #o_Zez_Reczny_Do_Nast;
      R     #o_Zez_Reczny_Do_Pop;
      R     #Help_H_Motor_Prawo;
      R     #Help_H_Motor_Lewo;
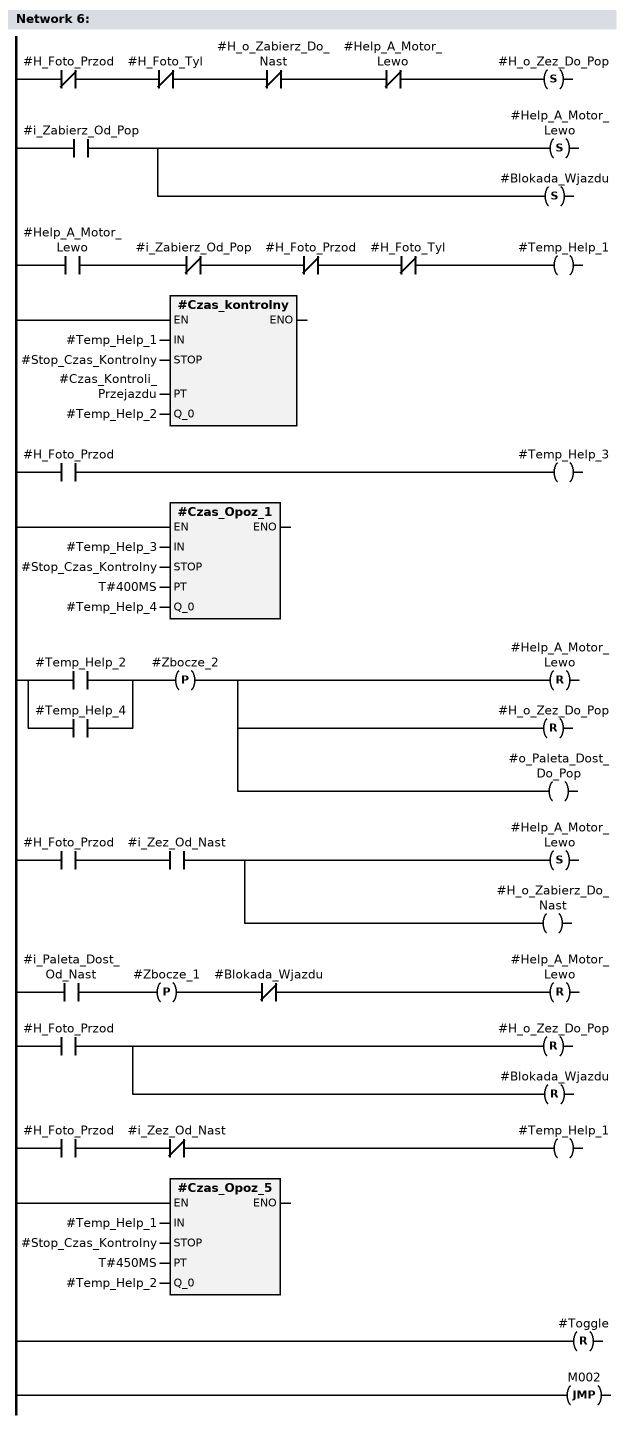
NETWORK
TITLE =
// Opis poszczegolnych krokow i skok do nich
// Tasma poprzednia pusta i bierzaca pusta
      AN    #H_Foto_Przod;
      AN    #H_Foto_Tyl;	//dodano bo hand
      AN    #H_o_Zabierz_Do_Nast;
      AN    #Help_A_Motor_Lewo;
      S     #H_o_Zez_Do_Pop;
      A     #i_Zabierz_Od_Pop;
      S     #Help_A_Motor_Lewo;
      S     #Blokada_Wjazdu;
//Warunek gdy pobranie z poprzedniej i miejsce foto srodek
//jest zajete
      A     #Help_A_Motor_Lewo;
      AN    #i_Zabierz_Od_Pop;
      AN    #H_Foto_Przod;
      AN    #H_Foto_Tyl;	//dodano bo hand
      =     #Temp_Help_1;
      CALL  #Czas_kontrolny (
           IN                       := #Temp_Help_1,
           STOP                     := #Stop_Czas_Kontrolny,
           PT                       := #Czas_Kontroli_Przejazdu,
           Q_0                      := #Temp_Help_2);
      A     #H_Foto_Przod;
//Paleta dostarczona
      =     #Temp_Help_3;
      CALL  #Czas_Opoz_1 (
           IN                       := #Temp_Help_3,
           STOP                     := #Stop_Czas_Kontrolny,
           PT                       := T#400MS,
           Q_0                      := #Temp_Help_4);
      A     #Temp_Help_2;
      O;
      A     #Temp_Help_4;
      FP    #Zbocze_2;
      R     #Help_A_Motor_Lewo;
      R     #H_o_Zez_Do_Pop;
      =     #o_Paleta_Dost_Do_Pop;
      A     #H_Foto_Przod;
      A     #i_Zez_Od_Nast;
//jest zezwolenie od nastepnej
      S     #Help_A_Motor_Lewo;
      =     #H_o_Zabierz_Do_Nast;
      A     #i_Paleta_Dost_Od_Nast;
      FP    #Zbocze_1;
//Potwierdzenie otrzymania palety
      AN    #Blokada_Wjazdu;
      R     #Help_A_Motor_Lewo;
      A     #H_Foto_Przod;
      R     #H_o_Zez_Do_Pop;
//Gdy zajete Foto_1 brak zezwolenia do poprzedniej
      R     #Blokada_Wjazdu;
      A     #H_Foto_Przod;
      AN    #i_Zez_Od_Nast;
//warunkowe zakonczenie pracy silnika gdy brak zezwolenia
//z nastepnej
      =     #Temp_Help_1;
      CALL  #Czas_Opoz_5 (
           IN                       := #Temp_Help_1,
           STOP                     := #Stop_Czas_Kontrolny,
           PT                       := T#450MS,
           Q_0                      := #Temp_Help_2);
      SET;
      R     #Toggle;
      JU    M002;
//wylacz toggle
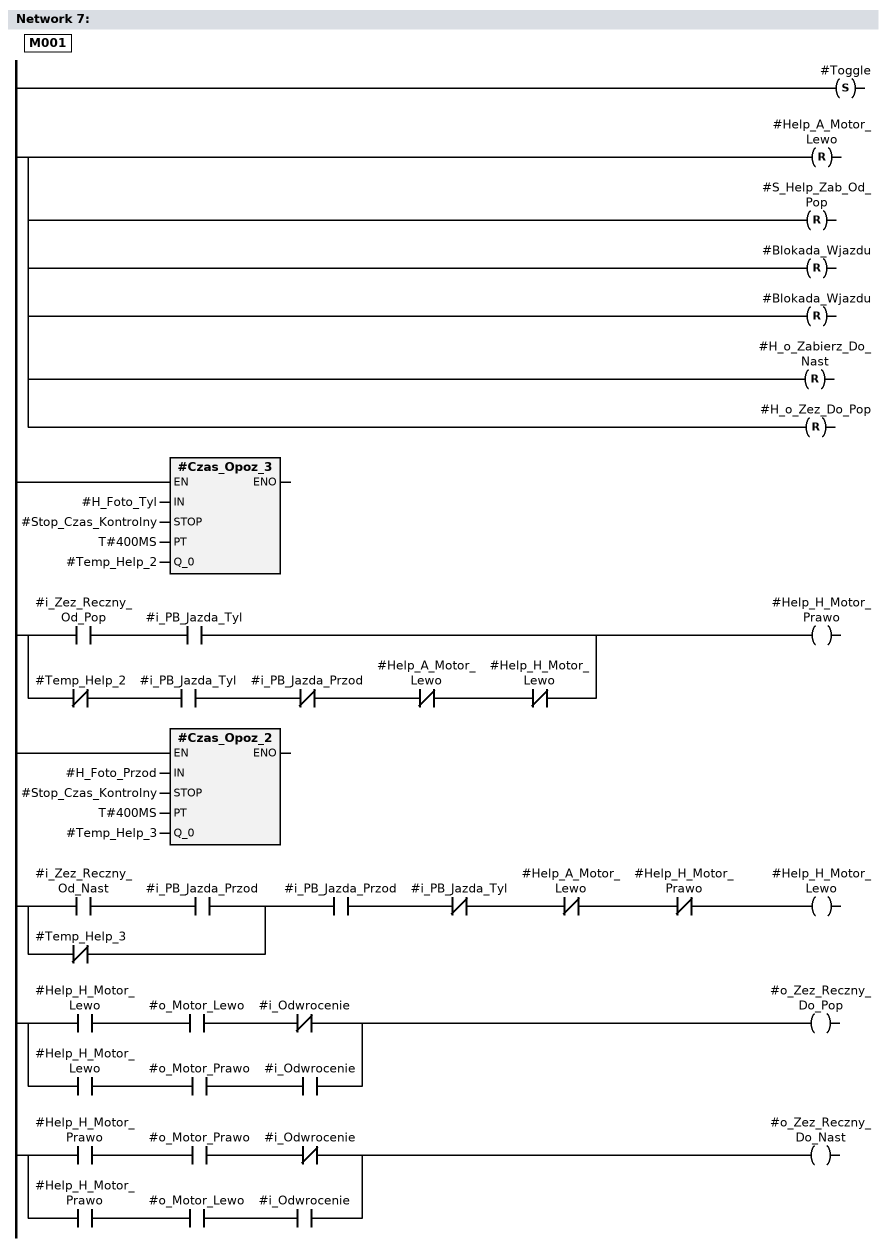
NETWORK
TITLE =
//Tryb reczny
//
M001: NOP   0;
//wlacz toggle
      SET;
      S     #Toggle;
//czyszczenie bitow z automatyki
      SET;
      R     #Help_A_Motor_Lewo;
      R     #S_Help_Zab_Od_Pop;
      R     #Blokada_Wjazdu;
      R     #Blokada_Wjazdu;
      R     #H_o_Zabierz_Do_Nast;
      R     #H_o_Zez_Do_Pop;
//ustawienie przyciskow
//jazda do tylu przycisk tyl
      CALL  #Czas_Opoz_3 (
           IN                       := #H_Foto_Tyl,
           STOP                     := #Stop_Czas_Kontrolny,
           PT                       := T#400MS,
           Q_0                      := #Temp_Help_2);
      A     #i_Zez_Reczny_Od_Pop;
      A     #i_PB_Jazda_Tyl;
      O;
      A(;
      AN    #Temp_Help_2;
      );
      A(;
      A     #i_PB_Jazda_Tyl;
      AN    #i_PB_Jazda_Przod;
      AN    #Help_A_Motor_Lewo;
      AN    #Help_H_Motor_Lewo;
      );
      =     #Help_H_Motor_Prawo;
//jazda do przodu
      CALL  #Czas_Opoz_2 (
           IN                       := #H_Foto_Przod,
           STOP                     := #Stop_Czas_Kontrolny,
           PT                       := T#400MS,
           Q_0                      := #Temp_Help_3);
      A(;
      A     #i_Zez_Reczny_Od_Nast;
      A     #i_PB_Jazda_Przod;
      O;
      AN    #Temp_Help_3;
      );
      A(;
      A     #i_PB_Jazda_Przod;
      AN    #i_PB_Jazda_Tyl;
      AN    #Help_A_Motor_Lewo;
      AN    #Help_H_Motor_Prawo;
      );
      =     #Help_H_Motor_Lewo;
      A     #Help_H_Motor_Lewo;
      A     #o_Motor_Lewo;
//wystawienie zezwolen do innych band wspolpracujacych recznie
//zezwolenie do tylu 
//zezwolenie do poprzedniej
      AN    #i_Odwrocenie;
      O;
      A     #Help_H_Motor_Lewo;
      A     #o_Motor_Prawo;
      A     #i_Odwrocenie;
      =     #o_Zez_Reczny_Do_Pop;
      A     #Help_H_Motor_Prawo;
      A     #o_Motor_Prawo;
//zezwolenie do nastepnej
      AN    #i_Odwrocenie;
      O;
      A     #Help_H_Motor_Prawo;
      A     #o_Motor_Lewo;
      A     #i_Odwrocenie;
      =     #o_Zez_Reczny_Do_Nast;
NETWORK
TITLE =
//Przypisanie wyjsc
//Koniec skoku
M002: NOP   0;
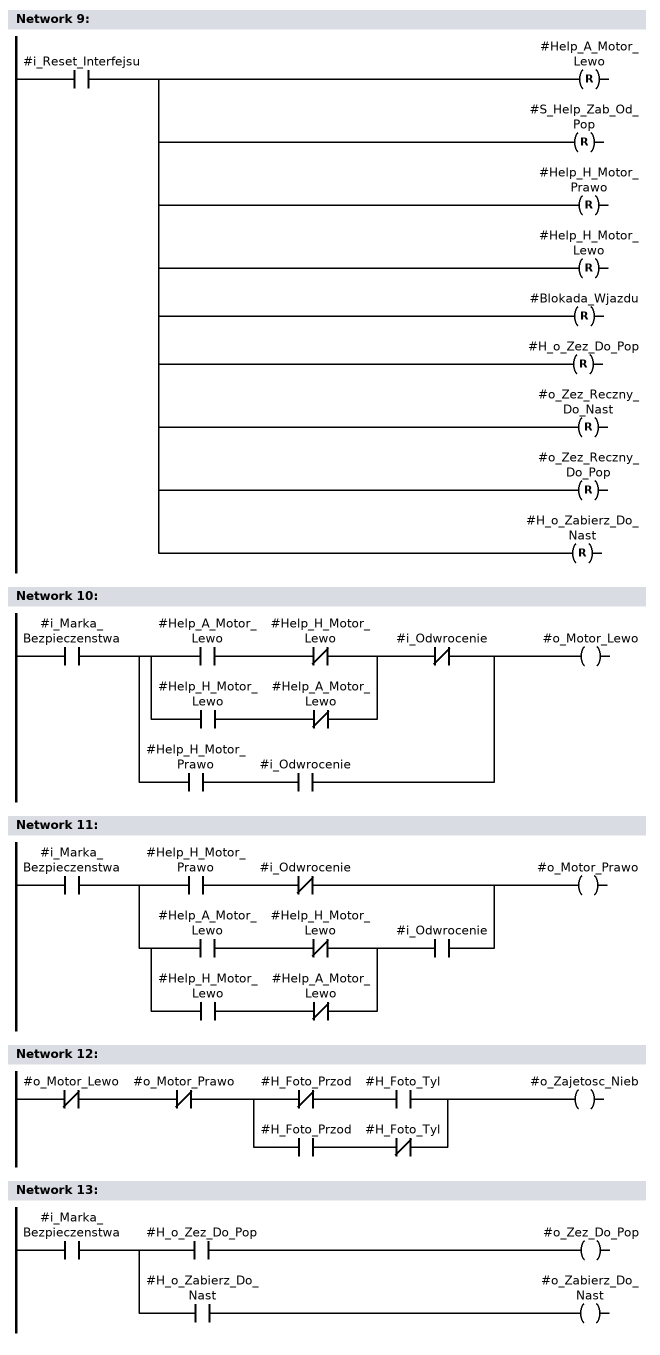
NETWORK
TITLE =
//Reset interfejsu
      A     #i_Reset_Interfejsu;
      R     #Help_A_Motor_Lewo;
      R     #S_Help_Zab_Od_Pop;
      R     #Help_H_Motor_Prawo;
      R     #Help_H_Motor_Lewo;
      R     #Blokada_Wjazdu;
      R     #H_o_Zez_Do_Pop;
      R     #o_Zez_Reczny_Do_Nast;
      R     #o_Zez_Reczny_Do_Pop;
      R     #H_o_Zabierz_Do_Nast;
NETWORK
TITLE =
////jazda automatyka reczny przod
      A     #i_Marka_Bezpieczenstwa;
      A(;
      A(;
      A     #Help_A_Motor_Lewo;
      AN    #Help_H_Motor_Lewo;
      O;
      A     #Help_H_Motor_Lewo;
      AN    #Help_A_Motor_Lewo;
      );
      AN    #i_Odwrocenie;
      O;
      A     #Help_H_Motor_Prawo;
      A     #i_Odwrocenie;
      );
      =     #o_Motor_Lewo;
NETWORK
TITLE =
////Jazda reczny tyl
      A     #i_Marka_Bezpieczenstwa;
      A(;
      A     #Help_H_Motor_Prawo;
      AN    #i_Odwrocenie;
      O;
      A(;
      A     #Help_A_Motor_Lewo;
      AN    #Help_H_Motor_Lewo;
      O;
      A     #Help_H_Motor_Lewo;
      AN    #Help_A_Motor_Lewo;
      );
      A     #i_Odwrocenie;
      );
      =     #o_Motor_Prawo;
NETWORK
TITLE =
//Zajetosc
      AN    #o_Motor_Lewo;
      AN    #o_Motor_Prawo;
      A(;
      AN    #H_Foto_Przod;
      A     #H_Foto_Tyl;
      O;
      A     #H_Foto_Przod;
      AN    #H_Foto_Tyl;
      );
      =     #o_Zajetosc_Nieb;
NETWORK
TITLE =
//Zezwolenie
      A     #i_Marka_Bezpieczenstwa;
      =     L 11.0;
      A     L 11.0;
      A     #H_o_Zez_Do_Pop;
      =     #o_Zez_Do_Pop;
      A     L 11.0;
      A     #H_o_Zabierz_Do_Nast;
      =     #o_Zabierz_Do_Nast;
NETWORK
TITLE =
//Koniec
//koniec
      BEU;
END_FUNCTION_BLOCK

FUNCTION_BLOCK "Banda_Poj_+_Tryb_Reczny"	// FB 33
//Funkcja realizujaca koncepcje bandy pojedycznej, ktora uwzglednia rowniez tryb 
//reczny. W celu lepszego sterowania trybem recznym nalezy do³o¿yæ:
//-fotokomorki na tyle bandy.
//-fotokomorka na tyle okresla rowniez zajetosc
//-jazda do tylu bandy mozliwa
//-jazda do przodu poza fotokomorke mozliwa gdy nastepna w ruchu i wolna.
//-do³o¿enie okresnia trybu reczny/auto gdzie auto to 1 
//
AUTHOR : Kng
FAMILY : Bandy
NAME : B_Single
VERSION : 1.0
VAR_INPUT
  i_Marka_Bezpieczenstwa : BOOL ;
  i_Rezerwa_1 : BOOL ;	//Zamrozenie stanu pracy
  i_Auto_Reczny : BOOL ;	//1-auto,0-reczny
  i_Foto_Przod : BOOL ;	//Foto na koncu tasmy
  i_Foto_Tyl : BOOL ;	//Foto zapobiegajace wyjechaniu palety do tylu
  i_Zez_Od_Nast : BOOL ;
  i_Paleta_Dost_Od_Nast : BOOL ;
  i_Zez_Reczny_Od_Nast : BOOL ;
  i_Zabierz_Od_Pop : BOOL ;
  i_Zez_Reczny_Od_Pop : BOOL ;
  i_PB_Jazda_Tyl : BOOL ;
  i_PB_Jazda_Przod : BOOL ;
  Czas_Kontroli_Przejazdu : TIME ;
END_VAR
VAR_OUTPUT
  o_Zabierz_Do_Nast : BOOL ;	//Rozkaz pobrania do nast bandy
  o_Zez_Do_Pop : BOOL ;
  o_Paleta_Dost_Do_Pop : BOOL ;
  o_Motor_Lewo : BOOL ;
  o_Motor_Prawo : BOOL ;
  o_Zez_Reczny_Do_Nast : BOOL ;
  o_Zez_Reczny_Do_Pop : BOOL ;
  o_Zajetosc_Nieb : BOOL ;	//Dla bezpieczenstwa transportu
END_VAR
VAR
  Czas_kontrolny : FB 21;
  Help_A_Motor_Lewo : BOOL ;
  S_Help_Zab_Od_Pop : BOOL ;
  Stop_Czas_Kontrolny : BOOL ;
  Zbocze_1 : BOOL ;
  Zbocze_2 : BOOL ;
  Blokada_Wjazdu : BOOL ;
  Help_H_Motor_Prawo : BOOL ;
  Help_H_Motor_Lewo : BOOL ;
  Toggle : BOOL ;	//bit przemienny dla auto i hand
  Help_8 : BOOL ;
  Help_9 : BOOL ;
END_VAR
VAR_TEMP
  Temp_Help_1 : BOOL ;
  Temp_Help_2 : BOOL ;
  Czas_zadany : TIME ;
  Czas_aktualny : TIME ;
END_VAR
BEGIN
NETWORK
TITLE =
//
// B1        B2         foto_1    foto_2         B5        B6
//(\\\\\\\\\\\\\\\\\\)  (\\\\\\\\\\\\\\\\\\)  (\\\\\\\\\\\\\\\\\\)
//                  M1                    M2                     M3
//         
//        zabierz <-- pobierz      |  zabierz    <--  pobierz  
//     zez_do_pop --> zez_od_nast  |  zez_od_pop -->  zez_od_nast
//                                  
//-Uklad dzielony jest na realizowane funkcje
//
//         <----------------------------------------- kierunek
//                  
//
// ten network celowo jest pusty
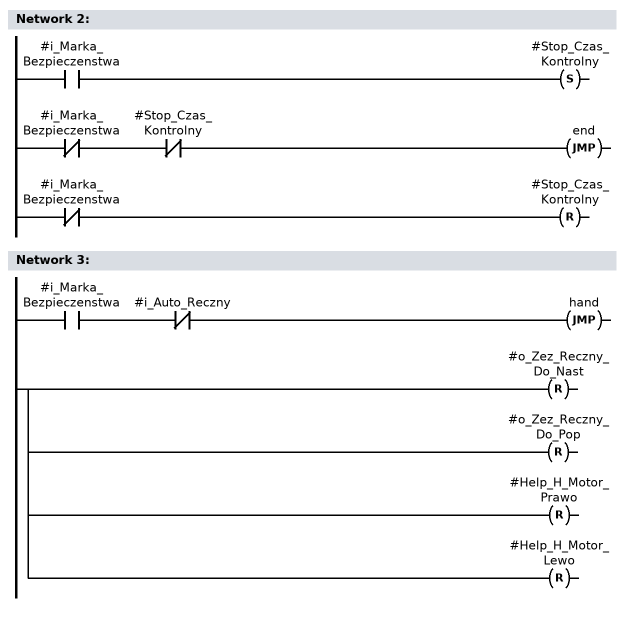
NETWORK
TITLE =
//Sprawdzenie stanu bezpieczenstwa lub freeze
//Skocz jezeli brak marki bezpieczenstwa
//Marka bezpieczenstwa ok gdy wysoki
      A     #i_Marka_Bezpieczenstwa;
      S     #Stop_Czas_Kontrolny;
      AN    #i_Marka_Bezpieczenstwa;
      AN    #Stop_Czas_Kontrolny;
      JC    end;
      AN    #i_Marka_Bezpieczenstwa;
      R     #Stop_Czas_Kontrolny;
NETWORK
TITLE =
//Wyznczenie zbocza pozytywnego i negatywnego
//skok do trybu recznego 
      A     #i_Marka_Bezpieczenstwa;
      AN    #i_Auto_Reczny;
      JC    hand;
//czyszczenie trybu recznego
      SET;
      R     #o_Zez_Reczny_Do_Nast;
      R     #o_Zez_Reczny_Do_Pop;
      R     #Help_H_Motor_Prawo;
      R     #Help_H_Motor_Lewo;
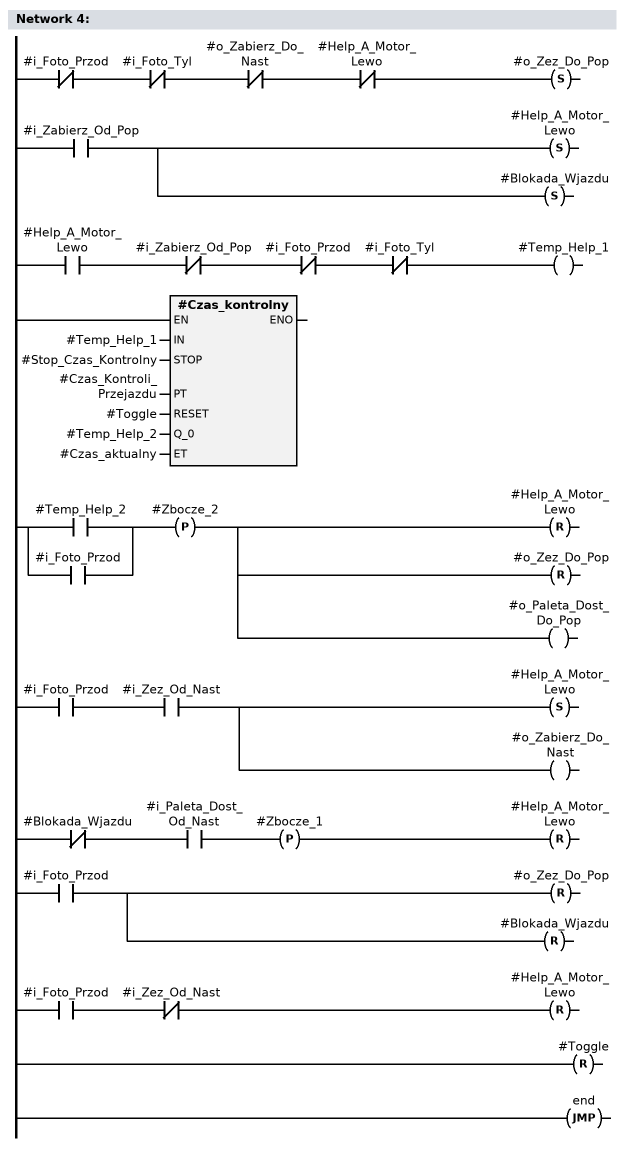
NETWORK
TITLE =
// Opis poszczegolnych krokow i skok do nich
// Tasma poprzednia pusta i bierzaca pusta
      AN    #i_Foto_Przod;
      AN    #i_Foto_Tyl;	//dodano bo hand
      AN    #o_Zabierz_Do_Nast;
      AN    #Help_A_Motor_Lewo;
      S     #o_Zez_Do_Pop;
      A     #i_Zabierz_Od_Pop;
      S     #Help_A_Motor_Lewo;
      S     #Blokada_Wjazdu;
//Warunek gdy pobranie z poprzedniej i miejsce foto srodek
//jest zajete
      A     #Help_A_Motor_Lewo;
      AN    #i_Zabierz_Od_Pop;
      AN    #i_Foto_Przod;
      AN    #i_Foto_Tyl;	//dodano bo hand
      =     #Temp_Help_1;
      CALL  #Czas_kontrolny (
           IN                       := #Temp_Help_1,
           STOP                     := #Stop_Czas_Kontrolny,
           PT                       := #Czas_Kontroli_Przejazdu,
           RESET                    := #Toggle,
           Q_0                      := #Temp_Help_2,
           ET                       := #Czas_aktualny);
//Paleta dostarczona
      A     #Temp_Help_2;
      O;
      A     #i_Foto_Przod;
      FP    #Zbocze_2;
      R     #Help_A_Motor_Lewo;
      R     #o_Zez_Do_Pop;
      =     #o_Paleta_Dost_Do_Pop;
//jest zezwolenie od nastepnej
      A     #i_Foto_Przod;
      A     #i_Zez_Od_Nast;
      S     #Help_A_Motor_Lewo;
      =     #o_Zabierz_Do_Nast;
//Potwierdzenie otrzymania palety
      AN    #Blokada_Wjazdu;
      A     #i_Paleta_Dost_Od_Nast;
      FP    #Zbocze_1;
      R     #Help_A_Motor_Lewo;
//Gdy zajete Foto_1 brak zezwolenia do poprzedniej
      A     #i_Foto_Przod;
      R     #o_Zez_Do_Pop;
      R     #Blokada_Wjazdu;
//warunkowe zakonczenie pracy silnika gdy brak zezwolenia
//z nastepnej
      A     #i_Foto_Przod;
      AN    #i_Zez_Od_Nast;
      R     #Help_A_Motor_Lewo;
//wylacz toggle
      SET;
      R     #Toggle;
//skocz do koniec
      JU    end;
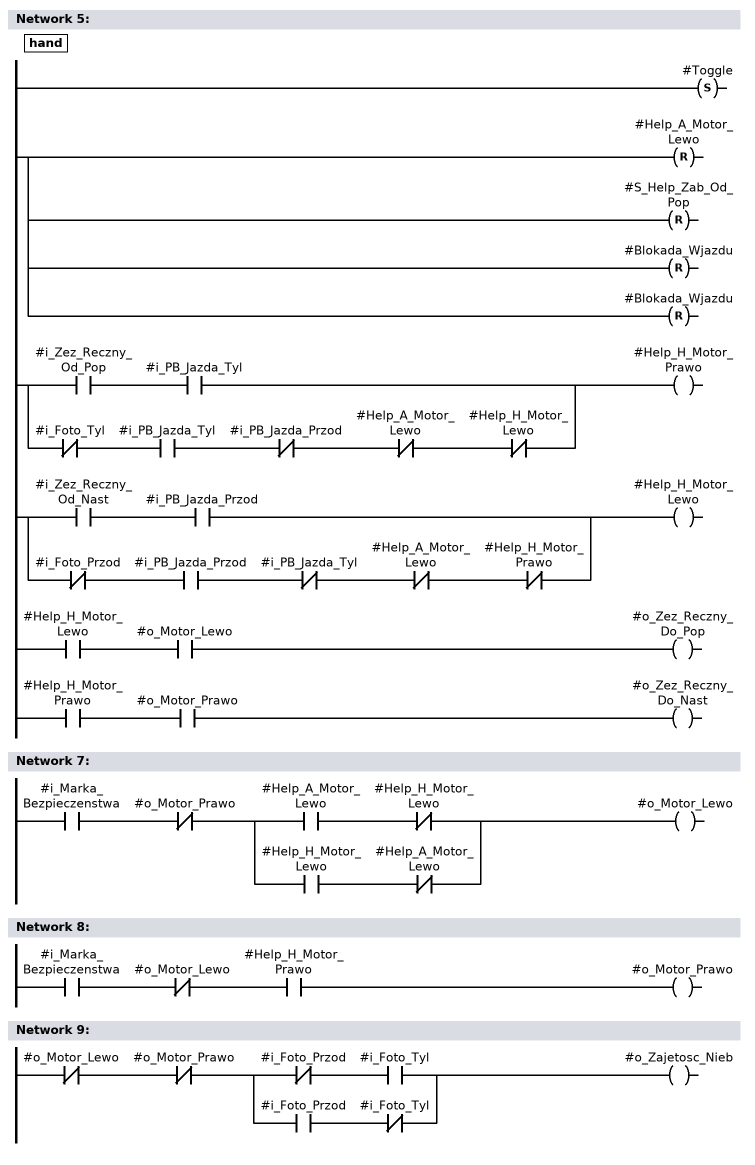
NETWORK
TITLE =
//Tryb reczny
//
hand: NOP   0;
//wlacz toggle
      SET;
      S     #Toggle;
//czyszczenie bitow z automatyki
      SET;
      R     #Help_A_Motor_Lewo;
      R     #S_Help_Zab_Od_Pop;
      R     #Blokada_Wjazdu;
      R     #Blokada_Wjazdu;
//ustawienie przyciskow
//jazda do tylu przycisk tyl
      A     #i_Zez_Reczny_Od_Pop;
      A     #i_PB_Jazda_Tyl;
      O;
      A(;
//      O     #i_Foto_Przod
      ON    #i_Foto_Tyl;
      );
      A(;
      A     #i_PB_Jazda_Tyl;
      AN    #i_PB_Jazda_Przod;
      AN    #Help_A_Motor_Lewo;
      AN    #Help_H_Motor_Lewo;
      );
      =     #Help_H_Motor_Prawo;
//jazda do przodu
      A     #i_Zez_Reczny_Od_Nast;
      A     #i_PB_Jazda_Przod;
      O;
      AN    #i_Foto_Przod;
      A(;
      A     #i_PB_Jazda_Przod;
      AN    #i_PB_Jazda_Tyl;
      AN    #Help_A_Motor_Lewo;
      AN    #Help_H_Motor_Prawo;
      );
      =     #Help_H_Motor_Lewo;
//wystawienie zezwolen do innych band wspolpracujacych recznie
//zezwolenie do tylu 
//zezwolenie do poprzedniej
      A     #Help_H_Motor_Lewo;
      A     #o_Motor_Lewo;
      =     #o_Zez_Reczny_Do_Pop;
//zezwolenie do nastepnej
      A     #Help_H_Motor_Prawo;
      A     #o_Motor_Prawo;
      =     #o_Zez_Reczny_Do_Nast;
NETWORK
TITLE =
//Przypisanie wyjsc
//Koniec skoku
end:  NOP   0;
NETWORK
TITLE =
////jazda automatyka reczny przod
      A     #i_Marka_Bezpieczenstwa;
      AN    #o_Motor_Prawo;
      A(;
      A     #Help_A_Motor_Lewo;
      AN    #Help_H_Motor_Lewo;
      O;
      A     #Help_H_Motor_Lewo;
      AN    #Help_A_Motor_Lewo;
      );
      =     #o_Motor_Lewo;
NETWORK
TITLE =
////Jazda reczny tyl
      A     #i_Marka_Bezpieczenstwa;
      AN    #o_Motor_Lewo;
      A     #Help_H_Motor_Prawo;
      =     #o_Motor_Prawo;
NETWORK
TITLE =
//Zajetosc
      AN    #o_Motor_Lewo;
      AN    #o_Motor_Prawo;
      A(;
      AN    #i_Foto_Przod;
      A     #i_Foto_Tyl;
      O;
      A     #i_Foto_Przod;
      AN    #i_Foto_Tyl;
      );
      =     #o_Zajetosc_Nieb;
NETWORK
TITLE =
//Koniec
//koniec
      BEU;
END_FUNCTION_BLOCK

FUNCTION_BLOCK "B_Obr_+_Reczny"	// FB 35
AUTHOR : Kng
FAMILY : Bandy
NAME : B_Obr
VERSION : 0.1
VAR_INPUT
  i_Marka_bezpieczenstwa : BOOL ;
  i_Tryb_Auto_Reczny : BOOL ;	//1-Auto;0-Rezczny
  i_Tryb_Uzbrajania : BOOL ;	//Paleta czeka na podwojny klik
  i_R_Zal_Uzbrajania : BOOL ;	//Zalaczenie Uzbrajania tylko w trybie recznym
  i_Uzbrajanie : BOOL ;	//Uzbrajanie jest aktywne
  i_Tryb_Inline : BOOL ;	//1-Paleta Prosto;0-Paleta w bok
  i_Foto_1 : BOOL ;
  i_Foto_2 : BOOL ;
  i_Zez_od_Wylot_1 : BOOL ;
  i_Zez_od_Wylot_2 : BOOL ;
  i_Paleta_Dost_Wylot_1 : BOOL ;
  i_Paleta_Dost_Wylot_2 : BOOL ;
  i_Zez_Reczny_Od_Wylot_1 : BOOL ;
  i_Zez_Reczny_Od_Wylot_2 : BOOL ;
  i_Zabierz_od_Wlot : BOOL ;
  i_Zez_Reczny_Od_Pop : BOOL ;
  i_PB_Jazda_CCW : BOOL ;
  i_PB_Jazda_CW : BOOL ;
  i_PB_Jazda_Przod : BOOL ;
  i_PB_Jazda_Tyl : BOOL ;
  i_PB_Pedal_Prawo : BOOL ;
  i_PB_Pedal_Lewo : BOOL ;
  i_czuj_poz_Wlot : BOOL ;
  i_czuj_ham_Wlot : BOOL ;
  i_czuj_poz_Wylot_2 : BOOL ;
  i_czuj_ham_Wylot_2 : BOOL ;
END_VAR
VAR_OUTPUT
  o_Paleta_Dost_Do_Wlot : BOOL ;
  o_Zabierz_do_Wylot_1 : BOOL ;
  o_Zabierz_do_Wylot_2 : BOOL ;
  o_Zez_Do_Wlot : BOOL ;
  o_Motor_1_lewo : BOOL ;
  o_Motor_1_prawo : BOOL ;
  o_Motor_1_Wolno : BOOL ;
  o_Motor_2_obr_s_Wylot_2 : BOOL ;	//Motor obrotnicy,kierunek strona wejscia,szybko
  o_Motor_2_obr_s_Wlot : BOOL ;	//Motor obrotnicy,kierunek strona wyjscia,szybko
  o_Motor_2_Wolno : BOOL ;	//Motor obrotnicy,kierunek strona wejscia,wolno
  o_Uzbrajanie_Aktywne : BOOL ;
  o_Zez_Reczny_do_Wlot : BOOL ;
  o_Zez_Reczny_do_Wylot_1 : BOOL ;
  o_Zez_Reczny_do_Wylot_2 : BOOL ;
END_VAR
VAR
  Kontrola_Rolki_Wlot : FB 20;
  Dojazd_Rolki_Wlot : FB 20;
  Opuszczenie_Bandy_Wlot_1 : FB 20;
  Opuszczenie_Bandy_Wlot_2 : FB 20;
  Sterowanie_Obrotem : FB 61;
  Silniki_nie_pracuja : BOOL ;
  Help_Motor_2_obr_Wylot_2 : BOOL ;	//Motor obrotnicy,kierunek strona wejscia,szybko
  Help_Motor_2_obr_Wlot : BOOL ;	//Motor obrotnicy,kierunek strona wyjscia,szybko
  Help_Motor_2_Wolno : BOOL ;	//Motor obrotnicy,kierunek strona wejscia,wolno
  Help_A_Motor_1_Lewo : BOOL ;
  Help_A_Motor_1_Prawo : BOOL ;
  Help_A_Motor_1_wolno : BOOL ;
  Help_H_Motor_1_Lewo : BOOL ;
  Help_H_Motor_1_Prawo : BOOL ;
  H_Edge_12 : BOOL ;
  H_Edge_13 : BOOL ;
  Stop_Czas_Kontrolny : BOOL ;
  H_Zez_do_Wlot : BOOL ;
  Pobranie_Wlot : BOOL ;
  H1_Doj_Rolki_Wlot : BOOL ;
  H2_Doj_Rolki_Wlot : BOOL ;
  T_Filtr_Rolki_Wlot : BOOL ;
  H_Paleta_Rowno_Na_Obr : BOOL ;
  H_Uzbroj_Palete : BOOL ;
  Tryb_Obrotnicy_Pelny : BOOL ;
  H_Obr_W_Kierunku_Wylotu : BOOL ;
  Obr_Na_Wlot : BOOL ;
  Obr_Na_Wylot_2 : BOOL ;
  Poz_Wlot : BOOL ;
  Poz_Wylot_2 : BOOL ;
  H_Oddanie_Do_Wylotu_1 : BOOL ;
  H_Oddanie_Do_Wylotu_2 : BOOL ;
  H_Powrot_Do_Wjazdu : BOOL ;
  H_Zabierz_do_Wylot_1 : BOOL ;
  H_Zabierz_do_Wylot_2 : BOOL ;
  H_Obracaj_W_Lewo : BOOL ;
  H_Obracaj_W_Prawo : BOOL ;
  H_Zez_na_Obr : BOOL ;
END_VAR
VAR_TEMP
  Temp_Help_1 : BOOL ;
  Temp_Help_2 : BOOL ;
  Czas_zadany : TIME ;
  Czas_aktualny : TIME ;
END_VAR
BEGIN
NETWORK
TITLE =
//                   
//Wlot                               Wylot_1
//()()()()|()()()()|  ()()()  |()()()()|()()()()
//()()()()|()()()()| ()()()() |()()()()|()()()()
//()()()()|()()()()| ()()()() |()()()()|()()()()
//()()()()|()()()()| ()()()() |()()()()|()()()()
//()()()()|()()()()|  ()()()  |()()()()|()()()()
//
//                  |()()()()|
//                  |()()()()|
//                  |()()()()| 
//                  |()()()()|
//                    Wylot_2
//         
//          pobierz --> zabierz   |     pobierz --> zabierz   
//     zez_od_nast <-- zez_do_pop | zez_od_nast <-- zez_od_pop
//                                  
//-Uklad dzielony jest na realizowane funkcje
//
//         
//                  
//
// ten network celowo jest pusty
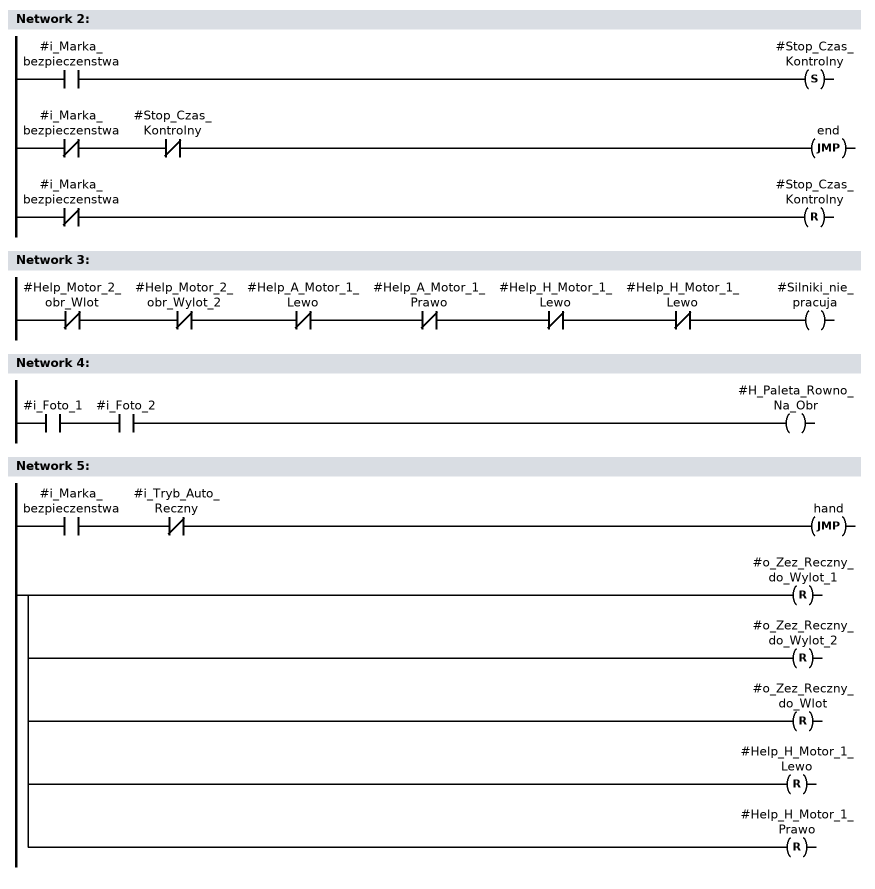
NETWORK
TITLE =
//Zatrzymanie uplywajacego czasu gdy brak bezpieczenstwa
//Skocz jezeli brak marki bezpieczenstwa
      A     #i_Marka_bezpieczenstwa;
      S     #Stop_Czas_Kontrolny;
      AN    #i_Marka_bezpieczenstwa;
      AN    #Stop_Czas_Kontrolny;
      JC    end;
      AN    #i_Marka_bezpieczenstwa;
      R     #Stop_Czas_Kontrolny;
NETWORK
TITLE =
//Sprawdzenie czy silniki nie pracuja
      AN    #Help_Motor_2_obr_Wlot;
      AN    #Help_Motor_2_obr_Wylot_2;
      AN    #Help_A_Motor_1_Lewo;
      AN    #Help_A_Motor_1_Prawo;
      AN    #Help_H_Motor_1_Lewo;
      AN    #Help_H_Motor_1_Lewo;
      =     #Silniki_nie_pracuja;
NETWORK
TITLE =
//Paleta rowno na obrotnicy
      A     #i_Foto_1;
      A     #i_Foto_2;
      =     #H_Paleta_Rowno_Na_Obr;
NETWORK
TITLE =
//Przejscie do trybu recznego
//skok do trybu recznego 
      A     #i_Marka_bezpieczenstwa;
      AN    #i_Tryb_Auto_Reczny;
      JC    hand;
//czyszczenie trybu recznego
      SET;
      R     #o_Zez_Reczny_do_Wylot_1;
      R     #o_Zez_Reczny_do_Wylot_2;
      R     #o_Zez_Reczny_do_Wlot;
      R     #Help_H_Motor_1_Lewo;
      R     #Help_H_Motor_1_Prawo;
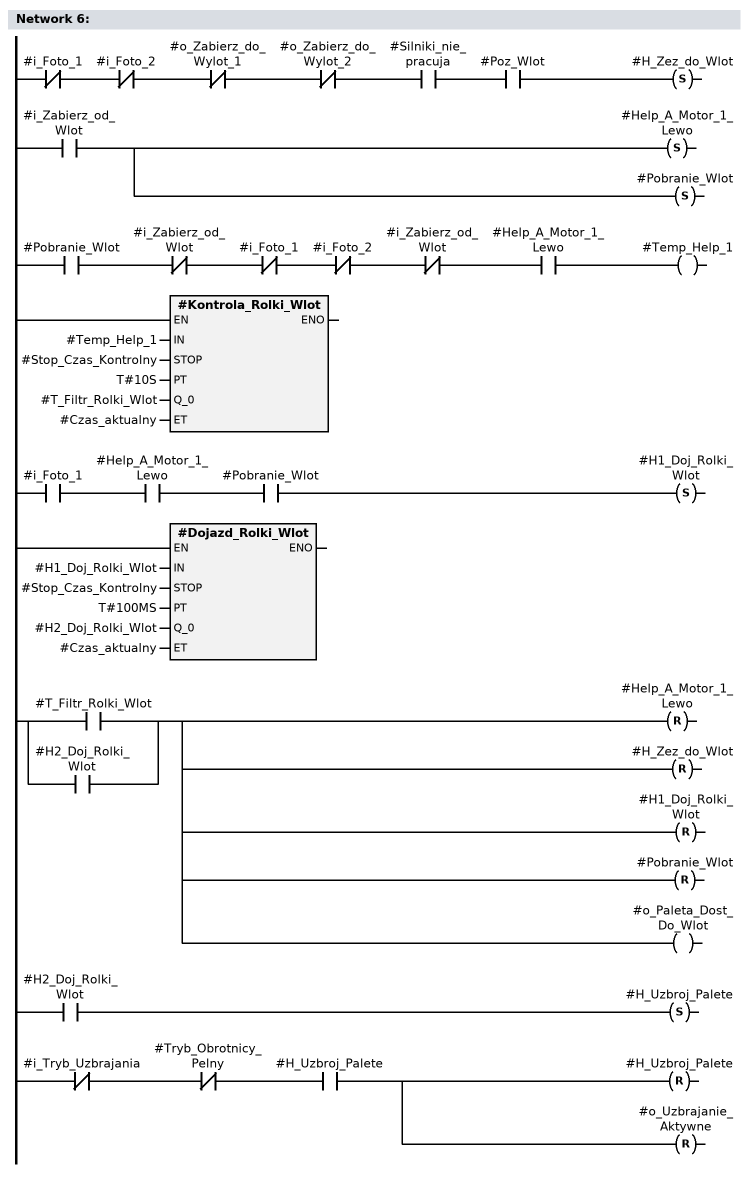
NETWORK
TITLE =
//Zezwolenie do porzedniej bandy (band segbertaf)
// Opis poszczegolnych krokow i skok do nich
// Tasma poprzednia pusta i bierzaca pusta
      AN    #i_Foto_1;
      AN    #i_Foto_2;
      AN    #o_Zabierz_do_Wylot_1;
      AN    #o_Zabierz_do_Wylot_2;
      A     #Silniki_nie_pracuja;
      A     #Poz_Wlot;
      S     #H_Zez_do_Wlot;
//gdy sygnal zabierz to blokada wjazdu
      A     #i_Zabierz_od_Wlot;
      S     #Help_A_Motor_1_Lewo;
      S     #Pobranie_Wlot;
//Czas kontrolny wjazdu na bande
      A     #Pobranie_Wlot;
      AN    #i_Zabierz_od_Wlot;
      AN    #i_Foto_1;
      AN    #i_Foto_2;
      AN    #i_Zabierz_od_Wlot;
      A     #Help_A_Motor_1_Lewo;
      =     #Temp_Help_1;
//Czas kontrolny dojazdu na stanowisko pracy
      CALL  #Kontrola_Rolki_Wlot (
           IN                       := #Temp_Help_1,
           STOP                     := #Stop_Czas_Kontrolny,
           PT                       := T#10S,
           Q_0                      := #T_Filtr_Rolki_Wlot,
           ET                       := #Czas_aktualny);
//Dojazd na pozycje na obrotnicy
      A     #i_Foto_1;
      A     #Help_A_Motor_1_Lewo;
      A     #Pobranie_Wlot;
      S     #H1_Doj_Rolki_Wlot;
      CALL  #Dojazd_Rolki_Wlot (
           IN                       := #H1_Doj_Rolki_Wlot,
           STOP                     := #Stop_Czas_Kontrolny,
           PT                       := T#100MS,
           Q_0                      := #H2_Doj_Rolki_Wlot,
           ET                       := #Czas_aktualny);
//Koniec pobierania palety z wlotu 1
      A     #T_Filtr_Rolki_Wlot;
      O;
      A     #H2_Doj_Rolki_Wlot;
      R     #Help_A_Motor_1_Lewo;
      R     #H_Zez_do_Wlot;
      R     #H1_Doj_Rolki_Wlot;
      R     #Pobranie_Wlot;
      =     #o_Paleta_Dost_Do_Wlot;
      A     #H2_Doj_Rolki_Wlot;
      S     #H_Uzbroj_Palete;
//Jezli wybrany tryb bez uzbrajania palety to
      AN    #i_Tryb_Uzbrajania;
      AN    #Tryb_Obrotnicy_Pelny;	//aby zapobiec zmianie w locie
      A     #H_Uzbroj_Palete;
      R     #H_Uzbroj_Palete;
      R     #o_Uzbrajanie_Aktywne;
//-------------------------------------------------
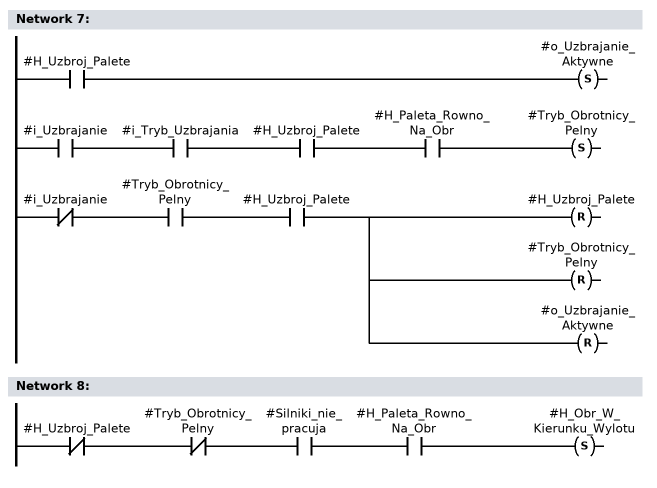
NETWORK
TITLE =
//Uzbrajanie Palety
//Rozpoczecie uzbrajania palety
//Sygnal uzbrojenie aktywne uruchamia funkcje aktywnego przycisku
      A     #H_Uzbroj_Palete;
      S     #o_Uzbrajanie_Aktywne;
//Aktywowanie funkcjonalnosci
      A     #i_Uzbrajanie;
      A     #i_Tryb_Uzbrajania;
      A     #H_Uzbroj_Palete;
      A     #H_Paleta_Rowno_Na_Obr;
      S     #Tryb_Obrotnicy_Pelny;
//Sygnal konca uzbrajania palety
      AN    #i_Uzbrajanie;
      A     #Tryb_Obrotnicy_Pelny;
      A     #H_Uzbroj_Palete;
      R     #H_Uzbroj_Palete;
      R     #Tryb_Obrotnicy_Pelny;
      R     #o_Uzbrajanie_Aktywne;
NETWORK
TITLE =
//Uzbojanie skonczone. Jazda na pozycje docelowa
//
      AN    #H_Uzbroj_Palete;
      AN    #Tryb_Obrotnicy_Pelny;
      A     #Silniki_nie_pracuja;
      A     #H_Paleta_Rowno_Na_Obr;
      S     #H_Obr_W_Kierunku_Wylotu;
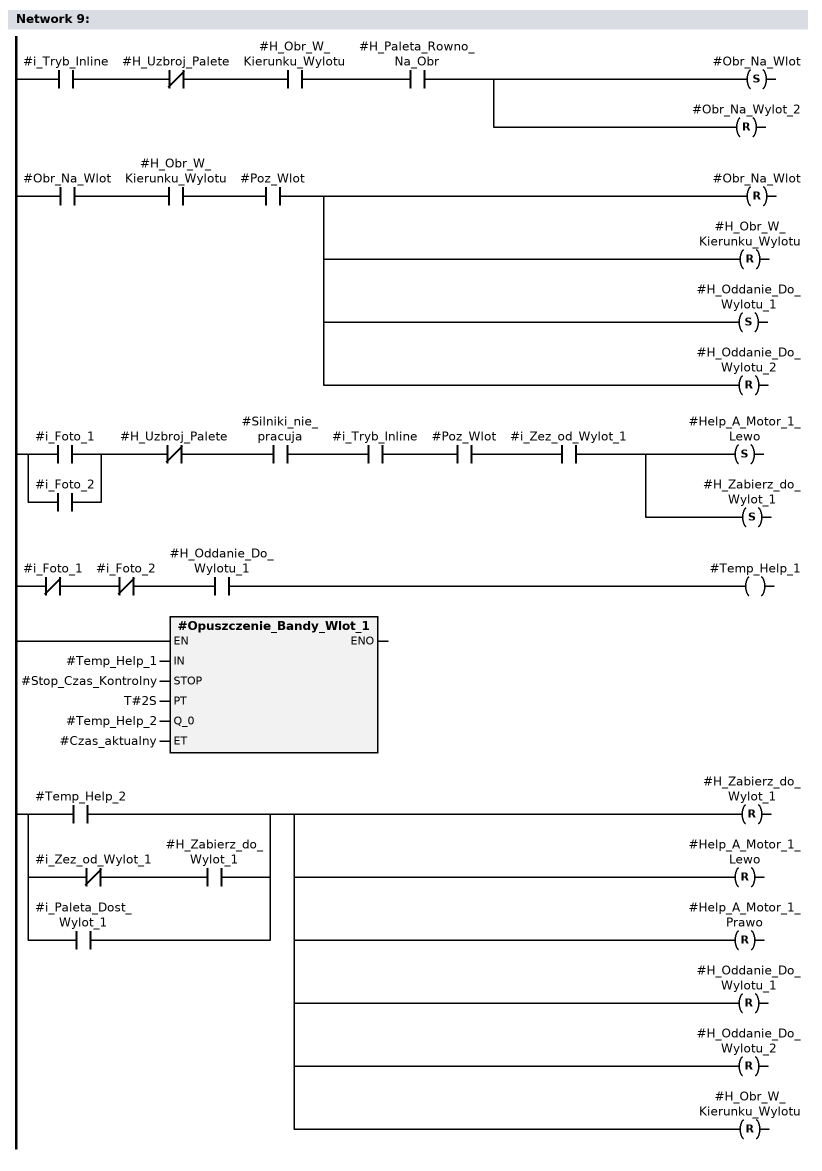
NETWORK
TITLE =
//Palet jedzie prosto tryb pracy inline
//
//Paleta ma wyjechac na wlot 1 (tryb pracy inline)
      A     #i_Tryb_Inline;
      AN    #H_Uzbroj_Palete;
      A     #H_Obr_W_Kierunku_Wylotu;
      A     #H_Paleta_Rowno_Na_Obr;
      S     #Obr_Na_Wlot;
      R     #Obr_Na_Wylot_2;
//-
      A     #Obr_Na_Wlot;
      A     #H_Obr_W_Kierunku_Wylotu;
      A     #Poz_Wlot;
      R     #Obr_Na_Wlot;
      R     #H_Obr_W_Kierunku_Wylotu;
      S     #H_Oddanie_Do_Wylotu_1;
      R     #H_Oddanie_Do_Wylotu_2;
//Oczekiwanie na zezwolenie
      O     #i_Foto_1;
      O     #i_Foto_2;
//      A     #H_Oddanie_Do_Wylotu_1
      AN    #H_Uzbroj_Palete;
      A     #Silniki_nie_pracuja;
      A     #i_Tryb_Inline;
      A     #Poz_Wlot;
      A     #i_Zez_od_Wylot_1;
      S     #Help_A_Motor_1_Lewo;
      S     #H_Zabierz_do_Wylot_1;
//reset sygnalu zabierz
      AN    #i_Foto_1;
      AN    #i_Foto_2;
      A     #H_Oddanie_Do_Wylotu_1;
      =     #Temp_Help_1;
      CALL  #Opuszczenie_Bandy_Wlot_1 (
           IN                       := #Temp_Help_1,
           STOP                     := #Stop_Czas_Kontrolny,
           PT                       := T#2S,
           Q_0                      := #Temp_Help_2,
           ET                       := #Czas_aktualny);
//koniec oddawania palety
      A     #Temp_Help_2;
      O;
      AN    #i_Zez_od_Wylot_1;
      A     #H_Zabierz_do_Wylot_1;
      O;
      A     #i_Paleta_Dost_Wylot_1;
      R     #H_Zabierz_do_Wylot_1;
      R     #Help_A_Motor_1_Lewo;
      R     #Help_A_Motor_1_Prawo;
      R     #H_Oddanie_Do_Wylotu_1;
      R     #H_Oddanie_Do_Wylotu_2;
      R     #H_Obr_W_Kierunku_Wylotu;
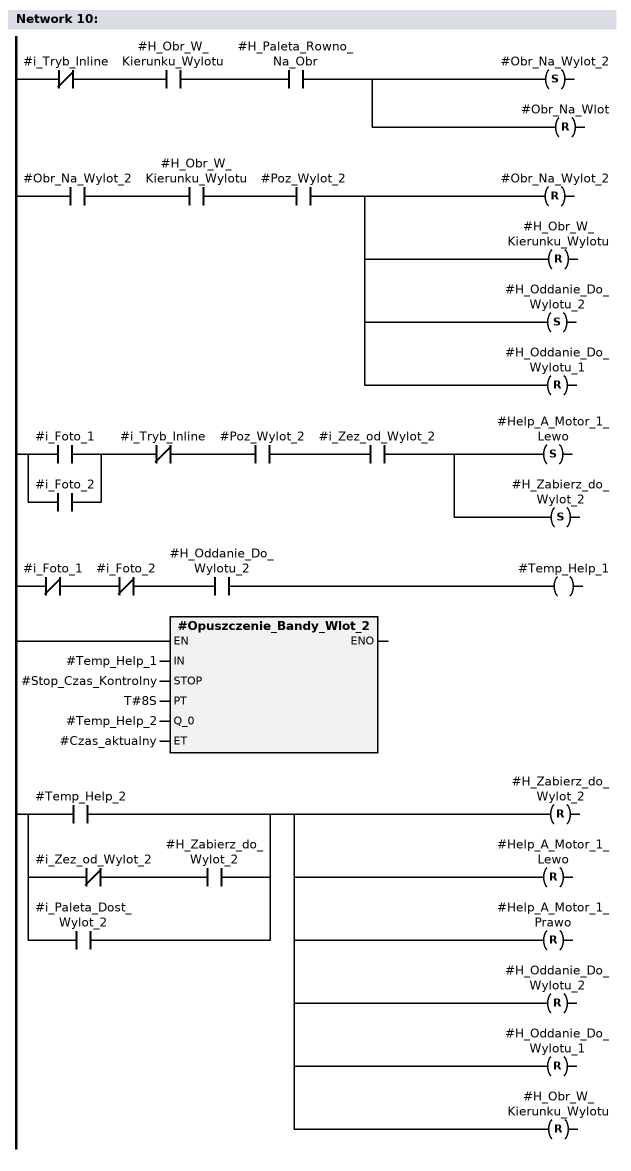
NETWORK
TITLE =
//Paleta jedzie w lewo 
//
//Paleta ma wyjechac na wylot 2  (tryb pracy inline)
      AN    #i_Tryb_Inline;
      A     #H_Obr_W_Kierunku_Wylotu;
      A     #H_Paleta_Rowno_Na_Obr;
      S     #Obr_Na_Wylot_2;
      R     #Obr_Na_Wlot;
      A     #Obr_Na_Wylot_2;
      A     #H_Obr_W_Kierunku_Wylotu;
      A     #Poz_Wylot_2;
      R     #Obr_Na_Wylot_2;
      R     #H_Obr_W_Kierunku_Wylotu;
      S     #H_Oddanie_Do_Wylotu_2;
      R     #H_Oddanie_Do_Wylotu_1;
//Oczekiwanie na zezwolenie
      O     #i_Foto_1;
      O     #i_Foto_2;
//   A     #H_Oddanie_Do_Wylotu_2
      AN    #i_Tryb_Inline;
      A     #Poz_Wylot_2;
      A     #i_Zez_od_Wylot_2;
      S     #Help_A_Motor_1_Lewo;
      S     #H_Zabierz_do_Wylot_2;
//reset sygnalu zabierz
      AN    #i_Foto_1;
      AN    #i_Foto_2;
      A     #H_Oddanie_Do_Wylotu_2;
      =     #Temp_Help_1;
      CALL  #Opuszczenie_Bandy_Wlot_2 (
           IN                       := #Temp_Help_1,
           STOP                     := #Stop_Czas_Kontrolny,
           PT                       := T#8S,
           Q_0                      := #Temp_Help_2,
           ET                       := #Czas_aktualny);
//koniece oddawania palety
      A     #Temp_Help_2;
      O;
      AN    #i_Zez_od_Wylot_2;
      A     #H_Zabierz_do_Wylot_2;
      O;
      A     #i_Paleta_Dost_Wylot_2;
      R     #H_Zabierz_do_Wylot_2;
      R     #Help_A_Motor_1_Lewo;
      R     #Help_A_Motor_1_Prawo;
      R     #H_Oddanie_Do_Wylotu_2;
      R     #H_Oddanie_Do_Wylotu_1;
      R     #H_Obr_W_Kierunku_Wylotu;
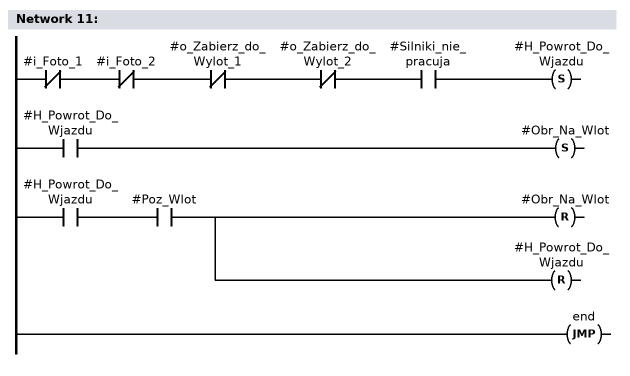
NETWORK
TITLE =
//Powrot obrotnicy na linie segberta
      AN    #i_Foto_1;
      AN    #i_Foto_2;
      AN    #o_Zabierz_do_Wylot_1;
      AN    #o_Zabierz_do_Wylot_2;
      A     #Silniki_nie_pracuja;
      S     #H_Powrot_Do_Wjazdu;
      A     #H_Powrot_Do_Wjazdu;
      S     #Obr_Na_Wlot;
      A     #H_Powrot_Do_Wjazdu;
      A     #Poz_Wlot;
      R     #Obr_Na_Wlot;
      R     #H_Powrot_Do_Wjazdu;
//Skocz na koniec programu
      JU    end;
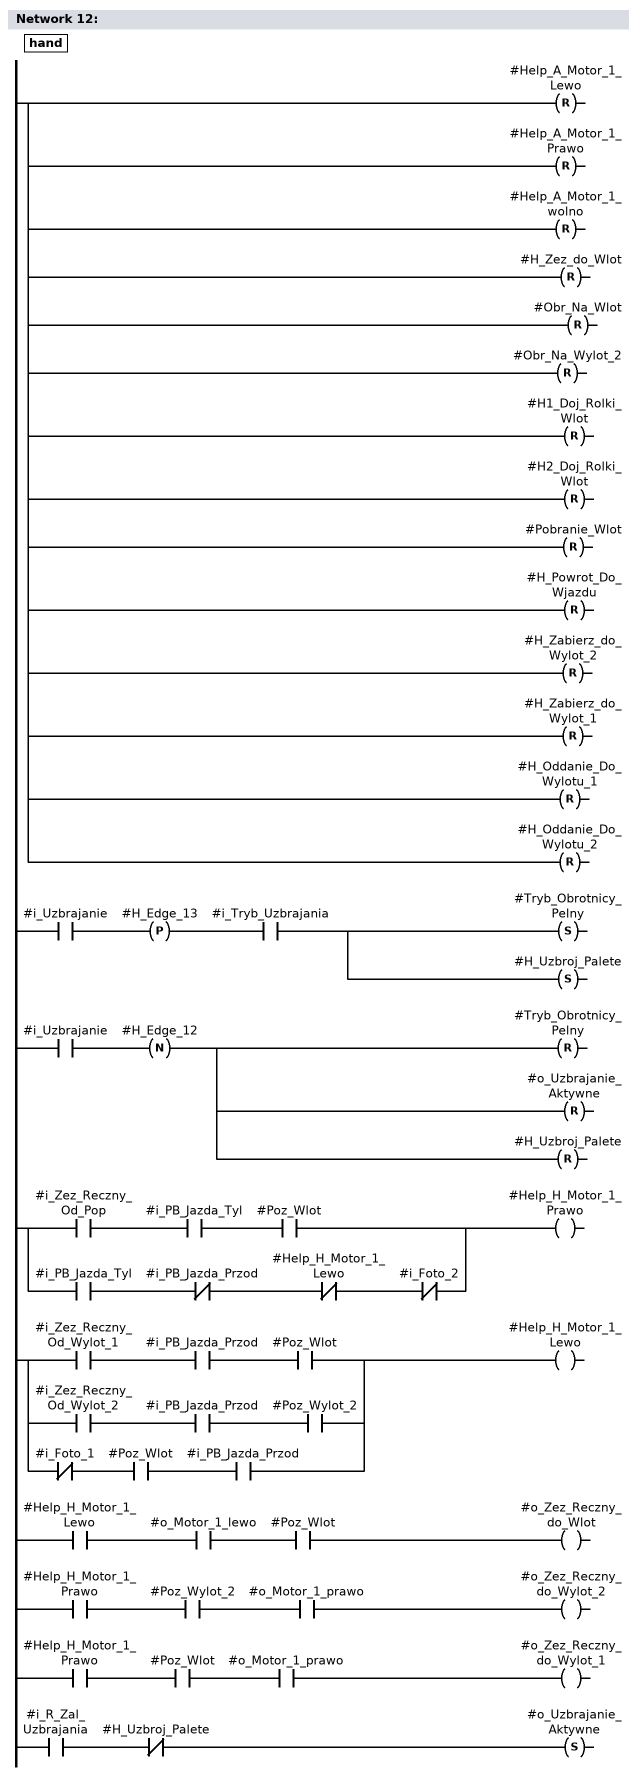
NETWORK
TITLE =
//Tryb reczny
//ustawienie przyciskow
//jazda do tylu przycisk tyl
hand: NOP   0;
//czyszczenie bitow z automatyki
      SET;
      R     #Help_A_Motor_1_Lewo;
      R     #Help_A_Motor_1_Prawo;
      R     #Help_A_Motor_1_wolno;
      R     #H_Zez_do_Wlot;
      R     #Obr_Na_Wlot;
      R     #Obr_Na_Wylot_2;
      R     #H1_Doj_Rolki_Wlot;
      R     #H2_Doj_Rolki_Wlot;
      R     #Pobranie_Wlot;
      R     #H_Powrot_Do_Wjazdu;
      R     #H_Zabierz_do_Wylot_2;
      R     #H_Zabierz_do_Wylot_1;
      R     #H_Oddanie_Do_Wylotu_1;
      R     #H_Oddanie_Do_Wylotu_2;
// Jezeli jest zalaczane uzbrajanie to mozna kontynuowac
      A     #i_Uzbrajanie;
      FP    #H_Edge_13;
      A     #i_Tryb_Uzbrajania;
      S     #Tryb_Obrotnicy_Pelny;
      S     #H_Uzbroj_Palete;
      A     #i_Uzbrajanie;
      FN    #H_Edge_12;
      R     #Tryb_Obrotnicy_Pelny;
      R     #o_Uzbrajanie_Aktywne;
      R     #H_Uzbroj_Palete;
//ustawienie przyciskow
//jazda do tylu przycisk tyl
      A     #i_Zez_Reczny_Od_Pop;
      A     #i_PB_Jazda_Tyl;
      A     #Poz_Wlot;
      O;
      A     #i_PB_Jazda_Tyl;
      AN    #i_PB_Jazda_Przod;
      AN    #Help_H_Motor_1_Lewo;
      AN    #i_Foto_2;
      =     #Help_H_Motor_1_Prawo;
//jazda do przodu
      A     #i_Zez_Reczny_Od_Wylot_1;
      A     #i_PB_Jazda_Przod;
      A     #Poz_Wlot;
      O;
      A     #i_Zez_Reczny_Od_Wylot_2;
      A     #i_PB_Jazda_Przod;
      A     #Poz_Wylot_2;
      O;
      AN    #i_Foto_1;
      A     #Poz_Wlot;
      A     #i_PB_Jazda_Przod;
      =     #Help_H_Motor_1_Lewo;
//wystawienie zezwolen do innych band wspolpracujacych recznie
//zezwolenie do tylu 
//zezwolenie do poprzedniej
      A     #Help_H_Motor_1_Lewo;
      A     #o_Motor_1_lewo;
      A     #Poz_Wlot;
      =     #o_Zez_Reczny_do_Wlot;
//zezwolenie do nastepnej
      A     #Help_H_Motor_1_Prawo;
      A     #Poz_Wylot_2;
      A     #o_Motor_1_prawo;
      =     #o_Zez_Reczny_do_Wylot_2;
      A     #Help_H_Motor_1_Prawo;
      A     #Poz_Wlot;
      A     #o_Motor_1_prawo;
      =     #o_Zez_Reczny_do_Wylot_1;
// Uzbrajanie palety  w trybier recznym
      A     #i_R_Zal_Uzbrajania;
      AN    #H_Uzbroj_Palete;
      S     #o_Uzbrajanie_Aktywne;
//skok do dalszej czesc programu
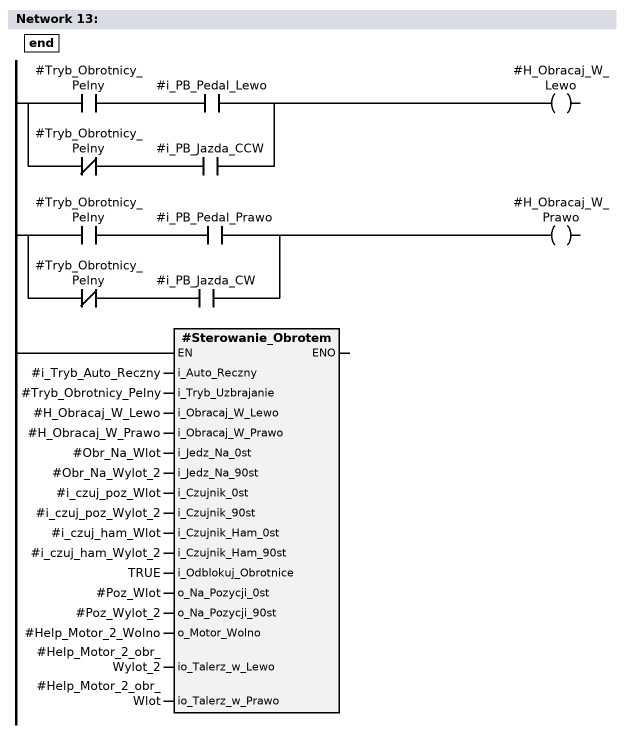
NETWORK
TITLE =
//Tryb obrotnicy pelny jest trybem dominujacym
end:  NOP   0;
      A     #Tryb_Obrotnicy_Pelny;
      A     #i_PB_Pedal_Lewo;
      O;
      AN    #Tryb_Obrotnicy_Pelny;
      A     #i_PB_Jazda_CCW;
      =     #H_Obracaj_W_Lewo;
      A     #Tryb_Obrotnicy_Pelny;
      A     #i_PB_Pedal_Prawo;
      O;
      AN    #Tryb_Obrotnicy_Pelny;
      A     #i_PB_Jazda_CW;
      =     #H_Obracaj_W_Prawo;
      CALL  #Sterowanie_Obrotem (
           i_Auto_Reczny            := #i_Tryb_Auto_Reczny,
           i_Tryb_Uzbrajanie        := #Tryb_Obrotnicy_Pelny,
           i_Obracaj_W_Lewo         := #H_Obracaj_W_Lewo,
           i_Obracaj_W_Prawo        := #H_Obracaj_W_Prawo,
           i_Jedz_Na_0st            := #Obr_Na_Wlot,
           i_Jedz_Na_90st           := #Obr_Na_Wylot_2,
           i_Czujnik_0st            := #i_czuj_poz_Wlot,
           i_Czujnik_90st           := #i_czuj_poz_Wylot_2,
           i_Czujnik_Ham_0st        := #i_czuj_ham_Wlot,
           i_Czujnik_Ham_90st       := #i_czuj_ham_Wylot_2,
           i_Odblokuj_Obrotnice     := TRUE,
           o_Na_Pozycji_0st         := #Poz_Wlot,
           o_Na_Pozycji_90st        := #Poz_Wylot_2,
           o_Motor_Wolno            := #Help_Motor_2_Wolno,
           io_Talerz_w_Lewo         := #Help_Motor_2_obr_Wylot_2,
           io_Talerz_w_Prawo        := #Help_Motor_2_obr_Wlot);
NETWORK
TITLE =
//Ten Network celowo wolny
